screen "fp_motor" 500x500
   on GenerateScreen: "show_tab"(1)
   IOField "I/O field_current" at 172,288 size 68x16; FormatPattern 999.9; Unit  A
      ProcessValue <- ".AO1b"
      Visibility <- ".FP_SHOW.AI1"
   IOField "I/O field_power" at 172,308 size 68x16; FormatPattern 999.9; Unit  kW
      ProcessValue <- ".AO2b"
      Visibility <- ".FP_SHOW.AI2"
   IOField "I/O field_rpm" at 172,328 size 68x16; FormatPattern 9999; Unit  rpm
      ProcessValue <- ".AO3b"
      Visibility <- ".FP_SHOW.AI3"
   IOField "I/O field_set_spd" at 84,356 size 68x16; FormatPattern 999.9; Unit  %
      ProcessValue <- ".SPSET"
      Visibility <- ".FP_SHOW.SP"
   Button "btn_md_auto" at 20,193 size 80x30; TextOff 'Auto'; Authorization "Operate"
      ObjectEnable <- ".FP_DIM.Auto"
      Visibility <- ".FP_SHOW.PB_Auto"
      Appearance <- ".ModePointer"
      on Click: SetBit(".FP_CMD.Auto")
   TextField "cntrl_box_cntrl_head" at 12,68 size 86x22; Text 'Start/Stop'
   Button "btn_md_loc" at 107,193 size 80x30; TextOff 'Local'; Authorization "Operate"
      ObjectEnable <- ".FP_DIM.Local"
      Visibility <- ".FP_SHOW.PB_Local"
      Appearance <- ".ModePointer"
      on Click: SetBit(".FP_CMD.Local")
   TextField "cntrl_box_model_head" at 12,164 size 49x22; Text 'Mode'
   Button "btn_md_man" at 195,193 size 80x30; TextOff 'Man'; Authorization "Operate"
      ObjectEnable <- ".FP_DIM.Manual"
      Visibility <- ".FP_SHOW.PB_Manual"
      Appearance <- ".ModePointer"
      on Click: SetBit(".FP_CMD.Manual")
   TextField "cntrl_box_am_text" at 20,288 size 47x17; Text 'Current'
      Visibility <- ".FP_SHOW.AI1"
   TextField "cntrl_box_am_text_1" at 20,308 size 38x17; Text 'Power'
      Visibility <- ".FP_SHOW.AI2"
   TextField "cntrl_box_model_head_1" at 12,260 size 162x22; Text 'Analog Measurment'
   TextField "cntrl_box_am_text_2" at 20,328 size 27x17; Text 'RPM'
      Visibility <- ".FP_SHOW.AI3"
   TextField "cntrl_box_am_text_3" at 20,355 size 16x17; Text 'SP'
      Visibility <- ".FP_SHOW.SP"
   IOField "I/O field_current_1" at 84,288 size 68x16; FormatPattern 999.9; Unit  %
      ProcessValue <- ".AO1a"
      Visibility <- ".FP_SHOW.AI1"
   IOField "I/O field_power_1" at 84,308 size 68x16; FormatPattern 999.9; Unit  %
      ProcessValue <- ".AO2a"
      Visibility <- ".FP_SHOW.AI2"
   IOField "I/O field_rpm_1" at 84,328 size 68x16; FormatPattern 999.9; Unit  %
      ProcessValue <- ".AO3a"
      Visibility <- ".FP_SHOW.AI3"
   Button "btn_satrt" at 20,100 size 80x30; TextOff 'Start'; Authorization "Operate"
      Visibility <- ".FP_SHOW.PB_Start1"
      ObjectEnable <- ".FP_DIM.Start1"
      on Click: SetBit(".FP_CMD.Start1")
   Button "btn_stop" at 300,100 size 80x30; TextOff 'Stop'; Authorization "Operate"
      Visibility <- ".FP_SHOW.PB_Stop"
      ObjectEnable <- ".FP_DIM.Stop"
      on Click: SetBit(".FP_CMD.Stop")
   TextField "header_txt" at 8,8 size 396x21; Text 'HEADER'
      Text <- ".DefaultText"
   SymbolicIOField "status I/O field_1" at 8,32 size 396x32; TextOn '1'; TextOff '0'; TextList "motor_status"
      ProcessValue <- ".StatusWork"
      Appearance <- ".StatusWork"
   SymbolicIOField "status I/O field_2" at 468,4 size 24x24; TextOn '1'; TextOff '0'; TextList "mode_l"
      ProcessValue <- ".ModePointer"
      Appearance <- ".ModePointer"
   Button "bt_tab_1" at 412,76 size 80x28; TextOff 'Control'
      on Click: "show_tab"(1)
   Button "bt_tab_3" at 412,139 size 80x28; TextOff 'Input'
      on Click: "show_tab"(3)
   Button "bt_tab_4" at 412,171 size 80x28; TextOff 'Output'
      on Click: "show_tab"(4)
   Button "bt_tab_5" at 412,203 size 80x28; TextOff 'Timers'
      on Click: "show_tab"(5)
   Button "bt_tab_6" at 412,235 size 80x28; TextOff 'Analog'
      on Click: "show_tab"(6)
   Button "bt_tab_7" at 412,267 size 80x28; TextOff 'Point para'
      on Click: "show_tab"(7)
   Button "bt_tab_8" at 412,299 size 80x28; TextOff 'Config'
      on Click: "show_tab"(8)
   Button "bt_tab_11" at 412,396 size 80x28; TextOff 'Info'
      on Click: "show_tab"(11)
   Button "bt_tab_12" at 412,428 size 80x28; TextOff 'Motion'
      on Click: "show_tab"(12)
      Visibility <- ".FP_SHOW.MD"
   Button "bt_tab_9" at 412,331 size 80x28; TextOff 'Config2'
      on Click: "show_tab"(9)
   Button "bt_tab_10" at 412,364 size 80x28; TextOff 'Diag'
      on Click: "show_tab"(10)
   Button "bt_tab_2" at 412,108 size 80x28; TextOff 'Interlock'
      on Click: "show_tab"(2)
   TextField "input_head" at 15,68 size 38x19; Text 'Input'
   TextField "input_rdy" at 24,96 size 200x20; Text 'RDY Ready'
   TextField "input_mcc" at 24,120 size 200x20; Text 'MCC MCC Ready'
   TextField "input_ovl" at 24,144 size 200x20; Text 'OVL Overload'
   TextField "input_ret1" at 24,168 size 200x20; Text 'RET1 Return'
   TextField "input_lstr1" at 24,192 size 200x20; Text 'LSTR1 Local Start'
   TextField "input_lstp" at 24,216 size 200x20; Text 'LSTP Local Stop'
   TextField "input_rem" at 24,240 size 200x20; Text 'REM Remote'
   TextField "input_ssw" at 24,264 size 200x20; Text 'SSW Safety Switch'
   TextField "input_es" at 24,288 size 200x20; Text 'ES Excessive Strt'
   TextField "input_tfaa" at 224,96 size 180x20; Text 'TFA Thermistor'
   TextField "input_drdy" at 225,120 size 180x20; Text 'DRDY Drv/MCC Rdy'
   TextField "input_stall" at 225,144 size 180x20; Text 'STALL Mtr Stalled'
   TextField "input_earth" at 225,168 size 180x20; Text 'EARTH Earth Fault'
   TextField "input_ubal" at 225,192 size 180x20; Text 'UBAL Crnt Unbal'
   TextField "input_gfa" at 224,216 size 180x20; Text 'GFA Gen Fault'
   TextField "input_gwa" at 224,240 size 180x20; Text 'GWA Gen Warn'
   TextField "input_busf" at 224,264 size 180x20; Text 'BUSF Bus Fault'
   TextField "input_dopr" at 224,288 size 180x20; Text 'DOPR Oper Posit'
   TextField "input_dtst" at 224,312 size 180x20; Text 'DTEST Test Pos'
   TextField "input_ack" at 224,336 size 180x20; Text 'ACK Reset Ack'
   TextField "input_head_1" at 202,68 size 106x19; Text 'Extend Input'
   TextField "input_head_2" at 13,352 size 96x19; Text 'Miscellaneous'
   TextField "input_sel" at 24,373 size 180x20; Text 'SEL Select'
   TextField "input_astr" at 24,396 size 200x20; Text 'ASTR Auto Start Req'
   IOField "status_bit_1g_0r_3" at 72,96 size 20x20; FormatPattern 1; Unit  
      ProcessValue <- ".DI.RDY"
      Appearance <- ".DI.RDY"
   IOField "status_bit_1g_0r_2" at 72,120 size 20x20; FormatPattern 1; Unit  
      ProcessValue <- ".DI.MCC"
      Appearance <- ".DI.MCC"
   IOField "status_bit_1g_0r_4" at 72,144 size 20x20; FormatPattern 1; Unit  
      ProcessValue <- ".DI.OVL"
      Appearance <- ".DI.OVL"
   IOField "status_bit_1grn_0gry_5" at 72,168 size 20x20; FormatPattern 1; Unit  
      ProcessValue <- ".DI.RET1"
      Appearance <- ".DI.RET1"
   IOField "status_bit_1grn_0gry_1" at 72,192 size 20x20; FormatPattern 1; Unit  
      ProcessValue <- ".DI.LSTR1"
      Appearance <- ".DI.LSTR1"
   IOField "status_bit_1g_0r_5" at 72,216 size 20x20; FormatPattern 1; Unit  
      ProcessValue <- ".DI.LSTP"
      Appearance <- ".DI.LSTP"
   IOField "status_bit_1g_0r_6" at 72,240 size 20x20; FormatPattern 1; Unit  
      ProcessValue <- ".DI.REM"
      Appearance <- ".DI.REM"
   IOField "status_bit_1g_0r_7" at 72,264 size 20x20; FormatPattern 1; Unit  
      Appearance <- ".DI.SSW"
      ProcessValue <- ".DI.SSW"
   IOField "status_bit_1g_0g_8" at 72,288 size 20x20; FormatPattern 1; Unit  
      ProcessValue <- ".DI.ES"
   IOField "status_bit_1g_0r_1" at 276,92 size 20x20; FormatPattern 1; Unit  
      ProcessValue <- ".DI.TFA"
      Appearance <- ".DI.TFA"
   IOField "status_bit_1g_0r_8" at 276,120 size 20x20; FormatPattern 1; Unit  
      ProcessValue <- ".DI.DRDY"
      Appearance <- ".DI.DRDY"
   IOField "status_bit_1g_0r_9" at 276,144 size 20x20; FormatPattern 1; Unit  
      ProcessValue <- ".DI.STALL"
      Appearance <- ".DI.STALL"
   IOField "status_bit_1g_0r_10" at 276,168 size 20x20; FormatPattern 1; Unit  
      ProcessValue <- ".DI.EARTH"
      Appearance <- ".DI.EARTH"
   IOField "status_bit_1g_0r_11" at 276,192 size 20x20; FormatPattern 1; Unit  
      ProcessValue <- ".DI.UBAL"
      Appearance <- ".DI.UBAL"
   IOField "status_bit_1g_0r_12" at 276,216 size 20x20; FormatPattern 1; Unit  
      ProcessValue <- ".DI.GFA"
      Appearance <- ".DI.GFA"
   IOField "status_bit_1g_0r_13" at 276,240 size 20x20; FormatPattern 1; Unit  
      ProcessValue <- ".DI.GWA"
      Appearance <- ".DI.GWA"
   IOField "status_bit_1g_0r_14" at 276,264 size 20x20; FormatPattern 1; Unit  
      ProcessValue <- ".DI.BUSF"
      Appearance <- ".DI.BUSF"
   IOField "status_bit_1g_0r_15" at 276,288 size 20x20; FormatPattern 1; Unit  
      ProcessValue <- ".DI.DOPR"
      Appearance <- ".DI.DOPR"
   IOField "status_bit_1grn_0gry_2" at 276,336 size 20x20; FormatPattern 1; Unit  
      ProcessValue <- ".DI.ACK"
      Appearance <- ".DI.ACK"
   IOField "status_bit_1red_0gry_3" at 276,312 size 20x20; FormatPattern 1; Unit  
      ProcessValue <- ".DI.DTEST"
      Appearance <- ".DI.DTEST"
   IOField "status_bit_1grn_0gry_3" at 72,373 size 20x20; FormatPattern 1; Unit  
      ProcessValue <- ".DI.SEL"
      Appearance <- ".DI.SEL"
   IOField "status_bit_1grn_0gry_4" at 72,396 size 20x20; FormatPattern 1; Unit  
      ProcessValue <- ".DI.ASTR"
      Appearance <- ".DI.ASTR"
   TextField "output_head_3" at 15,68 size 49x19; Text 'Output'
   TextField "output_ok_1" at 24,96 size 200x20; Text 'OK OK'
   TextField "output_sack_1" at 24,120 size 200x20; Text 'SACK Start Ack'
   TextField "output__rd1_1" at 24,144 size 200x20; Text 'RD1 Run Delay'
   TextField "output_run_1" at 24,168 size 200x20; Text 'RUN Run'
   TextField "output_con1_1" at 24,192 size 200x20; Text 'CON1 Command'
   TextField "input_tfaa_1" at 224,96 size 180x20; Text 'LOC Local'
   TextField "input_drdy_1" at 225,120 size 180x20; Text 'AUT Auto'
   TextField "input_stall_1" at 225,144 size 180x20; Text 'MAN Manual'
   TextField "input_earth_1" at 225,168 size 180x20; Text 'SS Single Strt'
   TextField "input_ubal_1" at 225,192 size 180x20; Text 'TESTP Test Pem'
   TextField "input_gfa_1" at 224,216 size 180x20; Text 'RES Reset'
   TextField "input_gwa_1" at 224,240 size 180x20; Text 'ASTW Start Warn'
   TextField "Output_head_4" at 202,68 size 114x19; Text 'Output Modes'
   TextField "output_head_5" at 13,291 size 38x19; Text 'Reset'
   IOField "status_bit_1g_0r_16" at 72,96 size 20x20; FormatPattern 1; Unit  
      ProcessValue <- ".DQ.OK"
      Appearance <- ".DQ.OK"
   IOField "status_bit_1g_0r_17" at 72,120 size 20x20; FormatPattern 1; Unit  
      ProcessValue <- ".DQ.SACK"
      Appearance <- ".DQ.SACK"
   IOField "status_bit_1g_0r_18" at 72,144 size 20x20; FormatPattern 1; Unit  
      ProcessValue <- ".DQ.RD1"
      Appearance <- ".DQ.RD1"
   IOField "status_bit_1grn_0gry_6" at 72,168 size 20x20; FormatPattern 1; Unit  
      ProcessValue <- ".DQ.RUN1"
      Appearance <- ".DQ.RUN1"
   IOField "status_bit_1grn_0gry_7" at 72,192 size 20x20; FormatPattern 1; Unit  
      ProcessValue <- ".DQ.CON1"
      Appearance <- ".DQ.CON1"
   IOField "status_bit_1g_0r_22" at 276,92 size 20x20; FormatPattern 1; Unit  
      ProcessValue <- ".DQ.LOC"
      Appearance <- ".DQ.LOC"
   IOField "status_bit_1g_0r_23" at 276,120 size 20x20; FormatPattern 1; Unit  
      ProcessValue <- ".DQ.AUT"
      Appearance <- ".DQ.AUT"
   IOField "status_bit_1g_0r_24" at 276,144 size 20x20; FormatPattern 1; Unit  
      ProcessValue <- ".DQ.MAN"
      Appearance <- ".DQ.MAN"
   IOField "status_bit_1g_0r_25" at 276,168 size 20x20; FormatPattern 1; Unit  
      ProcessValue <- ".DQ.SS"
      Appearance <- ".DQ.SS"
   IOField "status_bit_1g_0r_26" at 276,192 size 20x20; FormatPattern 1; Unit  
      ProcessValue <- ".DQ.TESTP"
      Appearance <- ".DQ.TESTP"
   IOField "status_bit_1g_0r_27" at 276,216 size 20x20; FormatPattern 1; Unit  
      ProcessValue <- ".DQ.RES"
      Appearance <- ".DQ.RES"
   IOField "status_bit_1g_0r_28" at 276,240 size 20x20; FormatPattern 1; Unit  
      ProcessValue <- ".DQ.ASTW"
      Appearance <- ".DQ.ASTW"
   Button "btn_reset" at 172,318 size 80x30; TextOff 'Reset'
      on Click: SetBit(".FP_CMD.Reset")
      ObjectEnable <- ".FP_DIM.Reset"
      Visibility <- ".FP_SHOW.PB_Reset"
   TextField "output_head_1" at 16,69 size 49x19; Text 'Timers'
   TextField "timers_text" at 24,96 size 100x20; Text 'Delay Start'
   IOField "delay_start_tm_sp" at 132,96 size 60x20; Authorization "User administration"; FormatPattern 9999; Unit  s
      ProcessValue <- ".FP_PARM.DelayStart_Pre"
   TextField "timers_text_1" at 24,120 size 100x20; Text 'Return M Tm'
   TextField "timers_text_2" at 24,144 size 100x20; Text 'Delayed Run'
   TextField "timers_text_3" at 24,168 size 100x20; Text 'Delayed Stop'
   TextField "timers_text_4" at 24,192 size 100x20; Text 'Start Warning'
   IOField "return_tm_sp" at 132,120 size 60x20; Authorization "User administration"; FormatPattern 9999; Unit  s
      ProcessValue <- ".FP_PARM.ReturnMon_Pre"
   IOField "delayed_run_tm_sp" at 132,144 size 60x20; Authorization "User administration"; FormatPattern 9999; Unit  s
      ProcessValue <- ".FP_PARM.RunDelay1_Pre"
   IOField "delay_stop_tm_sp" at 132,168 size 60x20; Authorization "User administration"; FormatPattern 999; Unit  s
      ProcessValue <- ".FP_PARM.DelayStop_Pre"
   IOField "delay_startsrm_tm_sp" at 132,192 size 60x20; Authorization "User administration"; FormatPattern 999; Unit  s
      ProcessValue <- ".FP_PARM.StartWarn_Pre"
   TextField "output_head_2" at 16,69 size 58x19; Text 'Current'
   TextField "analog_text_1" at 24,115 size 100x20; Text 'Minimum'
   IOField "ai1_min_sp" at 132,115 size 60x20; Authorization "User administration"; FormatPattern 9999.9; Unit  
      ProcessValue <- ".FP_PARM.AI1_Min"
   TextField "analog_text_2" at 147,93 size 33x17; Text 'Input'
   TextField "analog_text_3" at 223,93 size 44x17; Text 'Output'
   TextField "analog_text_4" at 303,93 size 36x17; Text 'Out:A'
   IOField "ao1a_min_sp" at 212,115 size 60x20; Authorization "User administration"; FormatPattern 9999.9; Unit  
      ProcessValue <- ".FP_PARM.AO1a_Min"
   IOField "ao1b_min_sp" at 292,115 size 60x20; Authorization "User administration"; FormatPattern 9999.9; Unit  
      ProcessValue <- ".FP_PARM.AO1b_Min"
   TextField "analog_text_5" at 24,139 size 100x20; Text 'Maximum'
   IOField "ai1_max_sp_1" at 132,139 size 60x20; Authorization "User administration"; FormatPattern 9999.9; Unit  
      ProcessValue <- ".FP_PARM.AI1_Max"
   IOField "ao1a_max_sp_1" at 212,139 size 60x20; Authorization "User administration"; FormatPattern 9999.9; Unit  
      ProcessValue <- ".FP_PARM.AO1a_Max"
   IOField "ao1b_max_sp_1" at 292,139 size 60x20; Authorization "User administration"; FormatPattern 9999.9; Unit  
      ProcessValue <- ".FP_PARM.AO1b_Max"
   IOField "ai1" at 132,167 size 60x20; FormatPattern 9999.9; Unit  
      ProcessValue <- ".AI1"
   IOField "ao1a" at 212,167 size 60x20; FormatPattern 9999.9; Unit  %
      ProcessValue <- ".AO1a"
   IOField "ao1b" at 292,167 size 60x20; FormatPattern 9999.9; Unit  A
      ProcessValue <- ".AO1b"
   TextField "output_head_6" at 15,196 size 49x19; Text 'Power'
   TextField "analog_text_6" at 23,243 size 100x20; Text 'Minimum'
   IOField "ai2_min_sp_1" at 131,243 size 60x20; Authorization "User administration"; FormatPattern 9999.9; Unit  
      ProcessValue <- ".FP_PARM.AI2_Min"
   TextField "analog_text_7" at 146,221 size 33x17; Text 'Input'
   TextField "analog_text_8" at 222,221 size 44x17; Text 'Output'
   TextField "analog_text_9" at 302,221 size 36x17; Text 'Out:A'
   IOField "ao2a_min_sp_1" at 211,243 size 60x20; Authorization "User administration"; FormatPattern 9999.9; Unit  
      ProcessValue <- ".FP_PARM.AO2a_Min"
   IOField "ao2b_min_sp_1" at 291,243 size 60x20; Authorization "User administration"; FormatPattern 9999.9; Unit  
      ProcessValue <- ".FP_PARM.AO2b_Min"
   TextField "analog_text_10" at 23,267 size 100x20; Text 'Maximum'
   IOField "ai2_max_sp_2" at 131,267 size 60x20; Authorization "User administration"; FormatPattern 9999.9; Unit  
      ProcessValue <- ".FP_PARM.AI2_Max"
   IOField "ao2a_max_sp_2" at 211,267 size 60x20; Authorization "User administration"; FormatPattern 9999.9; Unit  
      ProcessValue <- ".FP_PARM.AO2a_Max"
   IOField "ao2b_max_sp_2" at 291,267 size 60x20; Authorization "User administration"; FormatPattern 9999.9; Unit  
      ProcessValue <- ".FP_PARM.AO2b_Max"
   IOField "ai2_1" at 131,295 size 60x20; FormatPattern 9999.9; Unit  
      ProcessValue <- ".AI2"
   IOField "ao2a_1" at 211,295 size 60x20; FormatPattern 9999.9; Unit  %
      ProcessValue <- ".AO2a"
   IOField "ao2b_1" at 291,295 size 60x20; FormatPattern 9999.9; Unit  A
      ProcessValue <- ".AO2b"
   TextField "output_head_7" at 14,324 size 36x19; Text 'RPM'
   TextField "analog_text_11" at 23,372 size 100x20; Text 'Minimum'
   IOField "ai3_min_sp_2" at 131,372 size 60x20; Authorization "User administration"; FormatPattern 9999.9; Unit  
      ProcessValue <- ".FP_PARM.AI3_Min"
   TextField "analog_text_12" at 145,350 size 33x17; Text 'Input'
   TextField "analog_text_13" at 221,350 size 44x17; Text 'Output'
   TextField "analog_text_14" at 301,350 size 36x17; Text 'Out:A'
   IOField "ao3a_min_sp_2" at 211,372 size 60x20; Authorization "User administration"; FormatPattern 9999.9; Unit  
      ProcessValue <- ".FP_PARM.AO3a_Min"
   IOField "ao3b_min_sp_2" at 291,372 size 60x20; Authorization "User administration"; FormatPattern 9999.9; Unit  
      ProcessValue <- ".FP_PARM.AO3b_Min"
   TextField "analog_text_15" at 23,396 size 100x20; Text 'Maximum'
   IOField "ai3_max_sp_3" at 131,396 size 60x20; Authorization "User administration"; FormatPattern 9999.9; Unit  
      ProcessValue <- ".FP_PARM.AI3_Max"
   IOField "ao3a_max_sp_3" at 211,396 size 60x20; Authorization "User administration"; FormatPattern 9999.9; Unit  
      ProcessValue <- ".FP_PARM.AO3a_Max"
   IOField "ao3b_max_sp_3" at 291,396 size 60x20; Authorization "User administration"; FormatPattern 9999.9; Unit  
      ProcessValue <- ".FP_PARM.AO3b_Max"
   IOField "ai3_2" at 131,424 size 60x20; FormatPattern 9999.9; Unit  
      ProcessValue <- ".AI3"
   IOField "ao3a_2" at 211,424 size 60x20; FormatPattern 9999.9; Unit  %
      ProcessValue <- ".AO3a"
   IOField "ao3b_2" at 291,424 size 60x20; FormatPattern 9999.9; Unit  A
      ProcessValue <- ".AO3b"
   TextField "output_head_8" at 20,70 size 58x19; Text 'Current'
   CheckBox "Check box_1" at 28,96 size 180x20; Text0 'Alarm Supression'; Authorization "User administration"
   TextField "output_head_9" at 20,70 size 74x19; Text 'Unit Type'
   CheckBox "cb_Type_Indication" at 12,144 size 180x20; Text0 'Indication'; Authorization "User administration"
      ProcessValue <- ".FP_SEL.Type_Indication"
   OptionGroup "op_Type_Unimotor" at 12,96 size 180x20; Text0 'Uni directional motor'; Authorization "User administration"
      ProcessValue <- ".FP_SEL.Type_Unimotor"
   OptionGroup "op_Type_Bimotor" at 12,120 size 180x20; Text0 'Bi directional motor'; Authorization "User administration"
      ProcessValue <- ".FP_SEL.Type_Bimotor"
   CheckBox "cb_OutOfSevice" at 12,168 size 180x20; Text0 'Out of Sevices'; Authorization "User administration"
      ProcessValue <- ".FP_SEL.OutOfSevice"
   TextField "output_head_10" at 188,70 size 164x19; Text 'Start Warning Enable'
   CheckBox "cb_STW_Single" at 200,96 size 180x20; Text0 'Single Start'; Authorization "User administration"
      ProcessValue <- ".FP_SEL.STW_Single"
   CheckBox "cb_STW_Manual" at 200,120 size 180x20; Text0 'Manual'; Authorization "User administration"
      ProcessValue <- ".FP_SEL.STW_Manual"
   CheckBox "cb_STW_AutoStart" at 200,144 size 188x20; Text0 'Intrval Str (Auto Start)'; Authorization "User administration"
      ProcessValue <- ".FP_SEL.STW_AutoStart"
   CheckBox "cb_STW_Loca" at 200,168 size 188x20; Text0 'Local'; Authorization "User administration"
      ProcessValue <- ".FP_SEL.STW_Local"
   TextField "output_head_11" at 20,198 size 107x19; Text 'Alarm Handing'
   TextField "output_head_12" at 188,198 size 112x19; Text 'Enable Modes'
   CheckBox "Check box_8" at 12,224 size 180x20; Text0 'Warning Drive'; Authorization "User administration"
      ProcessValue <- ".FP_SEL.WarningDrive"
   CheckBox "Check box_9" at 12,248 size 180x20; Text0 'Sup by Parent Grp'; Authorization "User administration"
      ProcessValue <- ".FP_SEL.ParentSupress"
   CheckBox "Check box_10" at 12,272 size 188x20; Text0 'Pass Status to Par Grp'; Authorization "User administration"
      ProcessValue <- ".FP_SEL.ParentCollection"
   CheckBox "Check box_11" at 200,224 size 180x20; Text0 'Automatic'; Authorization "User administration"
      ProcessValue <- ".FP_EN.Mode_Auto"
   CheckBox "Check box_12" at 200,248 size 180x20; Text0 'Manual'; Authorization "User administration"
      ProcessValue <- ".FP_EN.Mode_Man"
   CheckBox "Check box_13" at 200,272 size 188x20; Text0 'Local'; Authorization "User administration"
      ProcessValue <- ".FP_EN.Mode_Loc"
   CheckBox "Check box_14" at 200,296 size 188x20; Text0 'Single Start FP'; Authorization "User administration"
      ProcessValue <- ".FP_EN.Mode_SS_FP"
   CheckBox "Check box_15" at 200,320 size 188x20; Text0 'Single Start Filed'; Authorization "User administration"
      ProcessValue <- ".FP_EN.Mode_SS_Field"
   CheckBox "Check box_16" at 200,344 size 188x20; Text0 'Test mode'; Authorization "User administration"
      ProcessValue <- ".FP_EN.Mode_Test"
   TextField "output_head_13" at 20,296 size 111x19; Text 'Enable Features'
   CheckBox "Check box_17" at 12,320 size 180x20; Text0 'Motion'; Authorization "User administration"
      ProcessValue <- ".FP_SEL.MD"
   CheckBox "Check box_18" at 12,344 size 180x20; Text0 'Motor Starter'; Authorization "User administration"
      ProcessValue <- ".FP_SEL.MotorStarter"
   CheckBox "Check box_19" at 12,368 size 188x20; Text0 'Quick Stop frm Unit'; Authorization "User administration"
      ProcessValue <- ".FP_EN.PB_QStop"
   CheckBox "Check box_20" at 12,392 size 188x20; Text0 'Reset Btn on Faceplate'; Authorization "User administration"
      ProcessValue <- ".FP_SHOW.PB_Reset"
   CheckBox "Check box_21" at 12,440 size 180x20; Text0 'Inch in Man Mode'; Authorization "User administration"
      ProcessValue <- ".FP_SEL.INCH_Man"
   CheckBox "Check box_22" at 12,464 size 180x20; Text0 'Inch in Loc Mode'; Authorization "User administration"
      ProcessValue <- ".FP_SEL.INCH_Loc"
   CheckBox "Check box_23" at 200,392 size 180x20; Text0 'Current'; Authorization "User administration"
      ProcessValue <- ".FP_SHOW.AI1"
   CheckBox "Check box_24" at 200,416 size 180x20; Text0 'Power'; Authorization "User administration"
      ProcessValue <- ".FP_SHOW.AI2"
   CheckBox "Check box_25" at 200,440 size 188x20; Text0 'RPM'; Authorization "User administration"
      ProcessValue <- ".FP_SHOW.AI3"
   CheckBox "Check box_26" at 200,464 size 188x20; Text0 'SP'; Authorization "User administration"
      ProcessValue <- ".FP_SHOW.SP"
   TextField "output_head_16" at 206,367 size 157x19; Text 'Display Analog Values'
   TextField "output_head_17" at 20,416 size 105x19; Text 'Inching Enable'
   TextField "output_head_14" at 20,70 size 98x19; Text 'Displat Inputs'
   CheckBox "cb_Type_Indication_1" at 204,300 size 100x20; Text0 'ASTRT'; Authorization "User administration"
      ProcessValue <- ".FP_SHOW.ASTR"
   CheckBox "cb_Type_Indication_2" at 16,100 size 100x192; Text0 'AI1'; Text1 'AI2'; Text2 'AI3'; Text3 'SP'; Text4 'MCC'; Text5 'RDY'; Text6 'OVL'; Text7 'LSTP'; Authorization "User administration"
      ProcessValue <- ".FP_SHOW.B1"
   CheckBox "cb_Type_Indication_3" at 108,100 size 100x192; Text6 'EARTH'; Text7 'UBAL'; Text4 'DRDY'; Text5 'STALL'; Text2 'ES'; Text3 'TFA'; Text0 'REM'; Text1 'SSW'; Authorization "User administration"
      ProcessValue <- ".FP_SHOW.B2"
   CheckBox "cb_Type_Indication_4" at 204,100 size 100x192; Text6 'LSTR1'; Text4 'DTEST'; Text5 'ACK'; Text2 'BUSF'; Text3 'DOPR'; Text0 'GFA'; Text1 'GWA'; Text7 'LSTR2'; Authorization "User administration"
      ProcessValue <- ".FP_SHOW.B3"
   TextField "output_head_15" at 15,68 size 114x19; Text 'PLC Subroutine'
   TextField "text_16" at 24,92 size 100x20; Text 'SubRoutine'
   TextField "text_1" at 24,120 size 100x20; Text 'Version'
   IOField "iof_vers" at 136,120 size 60x20; FormatPattern 9999; Unit  
      ProcessValue <- "[0]"
   TextField "text_2" at 24,148 size 100x20; Text 'Build'
   IOField "iof_build" at 136,148 size 60x20; FormatPattern 9999; Unit  
      ProcessValue <- "[1]"
   TextField "text_3" at 24,176 size 100x20; Text 'IOSys'
   TextField "output_head_18" at 212,68 size 129x19; Text 'Program Status'
   TextField "text_4" at 226,92 size 100x20; Text 'State Pointer'
   IOField "iof_state_pointer" at 338,92 size 60x20; FormatPattern 9999; Unit  
      ProcessValue <- ".BlockInfo[2]"
   TextField "text_5" at 227,120 size 100x20; Text 'State Pointer_Prev'
   IOField "iof_state_pointer_prev" at 339,120 size 60x20; FormatPattern 9999; Unit  
      ProcessValue <- ".BlockInfo[3]"
   TextField "output_head_19" at 16,228 size 106x19; Text 'PLC Reference'
   TextField "text_6" at 24,256 size 100x20; Text 'DB'
   IOField "iof_db" at 136,256 size 60x20; FormatPattern 9999; Unit  
      ProcessValue <- ".BlockInfo[4]"
   TextField "output_head_20" at 16,292 size 51x19; Text 'EcsRef'
   TextField "output_head_21" at 16,412 size 79x19; Text 'ParentInfo'
   TextField "text_7" at 24,320 size 100x20; Text 'FP Name'
   TextField "text_8" at 24,348 size 100x20; Text 'Blk Alg Ver'
   TextField "text_9" at 24,376 size 100x20; Text 'Status Alg Ver'
   IOField "parent_info" at 24,440 size 380x20; FormatPattern *; Unit  
      ProcessValue <- ".ParentInfo"
   TextField "interlockl_head_1" at 16,68 size 93x22; Text 'Interlocking'
   TextField "interlockl_head_2" at 12,225 size 174x22; Text 'Sequence Interlocking'
   TextField "interlockl_head_3" at 12,383 size 175x22; Text 'Sequence Stop Enable'
   TextField "interlock_1" at 28,100 size 140x20; Text 'Interlock 1'
      Text <- ".INTL01.DefaultText"
      Visibility <- ".INTL01"
   TextField "interlock_2" at 28,128 size 140x20; Text 'Interlock 2'
      Text <- ".INTL02.DefaultText"
      Visibility <- ".INTL04"
   TextField "interlock_3" at 28,156 size 140x20; Text 'Interlock 3'
      Text <- ".INTL03.DefaultText"
      Visibility <- ".INTL04"
   TextField "interlock_4" at 28,184 size 140x20; Text 'Interlock 4'
      Text <- ".INTL04.DefaultText"
      Visibility <- ".INTL04"
   TextField "STRT_1" at 28,256 size 140x20; Text 'Interlock 1'
      Visibility <- ".STR01"
      Text <- ".STR01.DefaultText"
   TextField "STRT_2" at 28,284 size 140x20; Text 'Interlock 2'
      Visibility <- ".STR02"
      Text <- ".STR02.DefaultText"
   TextField "STRT_3" at 28,312 size 140x20; Text 'Interlock 3'
      Visibility <- ".STR03"
      Text <- ".STR03.DefaultText"
   TextField "STRT_4" at 28,340 size 140x20; Text 'Interlock 4'
      Visibility <- ".STR04"
      Text <- ".STR04.DefaultText"
   SymbolicIOField "int_01" at 164,100 size 45x20; TextOn '1'; TextOff '0'; TextList "interlock_status_byte"
      ProcessValue <- ".INTL01"
      Appearance <- ".INTL01"
      Visibility <- ".INTL01"
   SymbolicIOField "int_2" at 164,128 size 45x20; TextOn '1'; TextOff '0'; TextList "interlock_status_byte"
      Visibility <- ".INTL02"
      ProcessValue <- ".INTL02"
      Appearance <- ".INTL02"
   SymbolicIOField "int_1" at 163,156 size 45x20; TextOn '1'; TextOff '0'; TextList "interlock_status_byte"
      ProcessValue <- ".INTL03"
      Visibility <- ".INTL03"
      Appearance <- ".INTL03"
   SymbolicIOField "int_3" at 164,184 size 45x20; TextOn '1'; TextOff '0'; TextList "interlock_status_byte"
      ProcessValue <- ".INTL04"
      Visibility <- ".INTL04"
      Appearance <- ".INTL04"
   TextField "interlock_5" at 221,100 size 140x20; Text 'Interlock 5'
      Text <- ".INTL05.DefaultText"
      Visibility <- ".INTL05"
   TextField "interlock_6" at 221,128 size 140x20; Text 'Interlock 6'
      Text <- ".INTL06.DefaultText"
      Visibility <- ".INTL06"
   TextField "interlock_7" at 221,156 size 140x20; Text 'Interlock 7'
      Text <- ".INTL07.DefaultText"
      Visibility <- ".INTL07"
   TextField "interlock_8" at 221,184 size 140x20; Text 'Interlock 8'
      Text <- ".INTL08.DefaultText"
      Visibility <- ".INTL08"
   SymbolicIOField "int_4" at 357,100 size 45x20; TextOn '1'; TextOff '0'; TextList "interlock_status_byte"
      Visibility <- ".INTL05"
      Appearance <- ".INTL05"
      ProcessValue <- ".INTL05"
   SymbolicIOField "int_5" at 357,128 size 45x20; TextOn '1'; TextOff '0'; TextList "interlock_status_byte"
      Visibility <- ".INTL06"
      Appearance <- ".INTL06"
      ProcessValue <- ".INTL06"
   SymbolicIOField "int_6" at 356,156 size 45x20; TextOn '1'; TextOff '0'; TextList "interlock_status_byte"
      Visibility <- ".INTL07"
      Appearance <- ".INTL07"
      ProcessValue <- ".INTL07"
   SymbolicIOField "int_7" at 357,184 size 45x20; TextOn '1'; TextOff '0'; TextList "interlock_status_byte"
      Visibility <- ".INTL08"
      Appearance <- ".INTL08"
      ProcessValue <- ".INTL08"
   SymbolicIOField "int_8" at 164,256 size 45x20; TextOn '1'; TextOff '0'; TextList "interlock_status_byte"
      Visibility <- ".STR01"
      Appearance <- ".STR01"
      ProcessValue <- ".STR01"
   SymbolicIOField "int_9" at 164,284 size 45x20; TextOn '1'; TextOff '0'; TextList "interlock_status_byte"
      Visibility <- ".STR02"
      Appearance <- ".STR02"
      ProcessValue <- ".STR02"
   SymbolicIOField "int_10" at 164,312 size 45x20; TextOn '1'; TextOff '0'; TextList "interlock_status_byte"
      Visibility <- ".STR03"
      Appearance <- ".STR03"
      ProcessValue <- ".STR03"
   SymbolicIOField "int_11" at 164,340 size 45x20; TextOn '1'; TextOff '0'; TextList "interlock_status_byte"
      Visibility <- ".STR04"
      Appearance <- ".STR04"
      ProcessValue <- ".STR04"
   TextField "STRT_5" at 221,256 size 140x20; Text 'Interlock 5'
      Visibility <- ".STR05"
      Text <- ".STR05.DefaultText"
   TextField "STRT_6" at 221,284 size 140x20; Text 'Interlock 6'
      Visibility <- ".STR06"
      Text <- ".STR05.DefaultText"
   TextField "STRT_7" at 221,312 size 140x20; Text 'Interlock 7'
      Visibility <- ".STR07"
      Text <- ".STR06.DefaultText"
   TextField "STRT_8" at 221,340 size 140x20; Text 'Interlock 8'
      Visibility <- ".STR08"
      Text <- ".STR08.DefaultText"
   SymbolicIOField "int_12" at 357,256 size 45x20; TextOn '1'; TextOff '0'; TextList "interlock_status_byte"
      Visibility <- ".STR05"
      Appearance <- ".STR05"
      ProcessValue <- ".STR05"
   SymbolicIOField "int_13" at 357,284 size 45x20; TextOn '1'; TextOff '0'; TextList "interlock_status_byte"
      Visibility <- ".STR06"
      Appearance <- ".STR06"
      ProcessValue <- ".STR06"
   SymbolicIOField "int_14" at 357,312 size 45x20; TextOn '1'; TextOff '0'; TextList "interlock_status_byte"
      Visibility <- ".STR07"
      Appearance <- ".STR07"
      ProcessValue <- ".STR07"
   SymbolicIOField "int_15" at 357,340 size 45x20; TextOn '1'; TextOff '0'; TextList "interlock_status_byte"
      Visibility <- ".STR08"
      Appearance <- ".STR08"
      ProcessValue <- ".STR08"
   TextField "STP_1" at 24,412 size 140x20; Text 'Interlock 1'
      Text <- ".STP01.DefaultText"
      Visibility <- ".STP01"
   TextField "STP_2" at 24,440 size 140x20; Text 'Interlock 2'
      Text <- ".STP02.DefaultText"
      Visibility <- ".STP02"
   TextField "STP_3" at 24,468 size 140x20; Text 'Interlock 3'
      Text <- ".STP03.DefaultText"
      Visibility <- ".STP03"
   SymbolicIOField "stp_int_1" at 160,412 size 45x20; TextOn '1'; TextOff '0'; TextList "interlock_status_byte"
      Visibility <- ".STP01"
      ProcessValue <- ".STP01"
      Appearance <- ".STP01"
   SymbolicIOField "stp_int_2" at 160,440 size 45x20; TextOn '1'; TextOff '0'; TextList "interlock_status_byte"
      Visibility <- ".STP02"
      ProcessValue <- ".STP01"
      Appearance <- ".STP02"
   SymbolicIOField "stp_int_3" at 160,468 size 45x20; TextOn '1'; TextOff '0'; TextList "interlock_status_byte"
      Visibility <- ".STP03"
      ProcessValue <- ".STP03"
      Appearance <- ".STP03"
   TextField "STP_4" at 220,412 size 140x20; Text 'Interlock 4'
      Visibility <- ".STP04"
      Text <- ".STP04.DefaultText"
   TextField "STP_5" at 220,440 size 140x20; Text 'Interlock 5'
      Visibility <- ".STP05"
      Text <- ".STP05.DefaultText"
   TextField "STP_6" at 220,468 size 140x20; Text 'Interlock 6'
      Visibility <- ".STP06"
      Text <- ".STP06.DefaultText"
   SymbolicIOField "stp_int_4" at 356,412 size 45x20; TextOn '1'; TextOff '0'; TextList "interlock_status_byte"
      Visibility <- ".STP04"
      Appearance <- ".STP04"
      ProcessValue <- ".STP04"
   SymbolicIOField "stp_int_5" at 356,440 size 45x20; TextOn '1'; TextOff '0'; TextList "interlock_status_byte"
      Visibility <- ".STP05"
      Appearance <- ".STP05"
      ProcessValue <- ".STP05"
   SymbolicIOField "stp_int_6" at 356,468 size 45x20; TextOn '1'; TextOff '0'; TextList "interlock_status_byte"
      Visibility <- ".STP06"
      Appearance <- ".STP06"
      ProcessValue <- ".STP06"

screen "Main.screen_window1" 0x0
   Siemens.Simatic.Hmi.Utah.GraphX.HmiScreenItem "Rectangle" at 0,0 size 0x0
   Siemens.Simatic.Hmi.Utah.GraphX.HmiScreenItem "header_txt" at 0,0 size 0x0

screen "fp_valve" 500x500
   on GenerateScreen: "show_tab"(1)
   Button "btn_md_auto" at 20,193 size 80x30; TextOff 'Auto'; Authorization "Operate"
      on Click: SetBit(".FP_CMD.Auto")
      Visibility <- ".FP_SHOW.PB_Auto"
      ObjectEnable <- ".FP_DIM.Auto"
      Appearance <- ".ModePointer"
   TextField "cntrl_box_cntrl_head" at 12,68 size 86x22; Text 'Start/Stop'
   Button "btn_md_loc" at 107,193 size 80x30; TextOff 'Local'; Authorization "Operate"
      on Click: SetBit(".FP_CMD.Local")
      Visibility <- ".FP_SHOW.PB_Local"
      ObjectEnable <- ".FP_DIM.Local"
      Appearance <- ".ModePointer"
   TextField "cntrl_box_model_head" at 12,164 size 49x22; Text 'Mode'
   Button "btn_md_man" at 195,193 size 80x30; TextOff 'Man'; Authorization "Operate"
      on Click: SetBit(".FP_CMD.Manual")
      Visibility <- ".FP_SHOW.PB_Manual"
      ObjectEnable <- ".FP_DIM.Manual"
      Appearance <- ".ModePointer"
   Button "btn_open" at 20,100 size 80x30; TextOff 'Open'; Authorization "Operate"
      on Click: SetBit(".FP_CMD.Start1")
      Visibility <- ".FP_SHOW.PB_Start1"
      ObjectEnable <- ".FP_DIM.Start1"
   Button "btn_close" at 300,100 size 80x30; TextOff 'Close'; Authorization "Operate"
      on Click: SetBit(".FP_CMD.Start2")
      ObjectEnable <- ".FP_DIM.Start2"
      Visibility <- ".FP_SHOW.PB_Start2"
   Button "btn_stop" at 156,128 size 80x30; TextOff 'Stop'; Authorization "Operate"
      on Click: SetBit(".FP_CMD.Stop")
      Visibility <- ".FP_SHOW.PB_Stop"
      ObjectEnable <- ".FP_DIM.Stop"
   TextField "header_txt" at 8,8 size 396x21; Text 'HEADER'
      Text <- ".DefaultText"
   SymbolicIOField "status I/O field_2" at 468,4 size 24x24; TextOn '1'; TextOff '0'; TextList "mode_l"
      ProcessValue <- ".ModePointer"
      Appearance <- ".ModePointer"
   Button "bt_tab_1" at 412,76 size 80x28; TextOff 'Control'
      on Click: "show_tab"(1)
   Button "bt_tab_3" at 412,139 size 80x28; TextOff 'Input'
      on Click: "show_tab"(3)
   Button "bt_tab_4" at 412,171 size 80x28; TextOff 'Output'
      on Click: "show_tab"(4)
   Button "bt_tab_5" at 412,203 size 80x28; TextOff 'Timers'
      on Click: "show_tab"(5)
   Button "bt_tab_7" at 412,234 size 80x28; TextOff 'Point para'
      on Click: "show_tab"(7)
   Button "bt_tab_8" at 412,266 size 80x28; TextOff 'Config'
      on Click: "show_tab"(8)
   Button "bt_tab_11" at 412,330 size 80x28; TextOff 'Info'
      on Click: "show_tab"(11)
   Button "bt_tab_9" at 412,298 size 80x28; TextOff 'Config2'
      on Click: "show_tab"(9)
   Button "bt_tab_2" at 412,108 size 80x28; TextOff 'Interlock'
      on Click: "show_tab"(2)
   SymbolicIOField "status I/O field_1" at 124,32 size 165x29; TextOn '1'; TextOff '0'; TextList "valve_status"
      ProcessValue <- ".StatusWork"
      Appearance <- ".StatusWork"
   TextField "input_head" at 15,68 size 38x19; Text 'Input'
   TextField "input_rdy" at 24,96 size 200x20; Text 'RDY Ready'
   TextField "input_ovl" at 24,120 size 200x20; Text 'OVL Overload'
   TextField "input_lstr1" at 24,144 size 200x20; Text 'LSP1 Lim Pos Open'
   TextField "input_lstp" at 24,168 size 200x20; Text 'LSP2 Lim Pos Close'
   TextField "input_rem" at 24,240 size 200x20; Text 'REM Remote'
   TextField "input_ssw" at 24,264 size 200x20; Text 'SSW Safety Switch'
   TextField "input_drdy" at 225,97 size 180x20; Text 'DRDY Drv/MCC Rdy'
   TextField "input_gfa" at 224,121 size 180x20; Text 'GFA Gen Fault'
   TextField "input_gwa" at 224,145 size 180x20; Text 'GWA Gen Warn'
   TextField "input_busf" at 224,169 size 180x20; Text 'BUSF Bus Fault'
   TextField "input_dtst" at 224,193 size 180x20; Text 'UTEST Test Pos'
   TextField "input_head_1" at 202,68 size 106x19; Text 'Extend Input'
   TextField "input_head_2" at 13,352 size 96x19; Text 'Miscellaneous'
   TextField "input_sel" at 24,376 size 180x20; Text 'SEL Select'
   IOField "status_bit_1g_0r_3" at 72,96 size 20x20; FormatPattern 1; Unit  
      ProcessValue <- ".DI.RDY"
      Appearance <- ".DI.RDY"
   IOField "status_bit_1g_0r_4" at 72,120 size 20x20; FormatPattern 1; Unit  
      ProcessValue <- ".DI.OVL"
      Appearance <- ".DI.OVL"
   IOField "status_bit_1grn_0gry_1" at 72,144 size 20x20; FormatPattern 1; Unit  
      Appearance <- ".DI.LSP1"
      ProcessValue <- ".DI.LSP1"
   IOField "status_bit_1g_0r_5" at 72,168 size 20x20; FormatPattern 1; Unit  
      Appearance <- ".DI.LSP2"
      ProcessValue <- ".DI.LSP2"
   IOField "status_bit_1g_0r_6" at 72,240 size 20x20; FormatPattern 1; Unit  
      ProcessValue <- ".DI.REM"
      Appearance <- ".DI.REM"
   IOField "status_bit_1g_0r_7" at 72,264 size 20x20; FormatPattern 1; Unit  
      ProcessValue <- ".DI.SSW"
      Appearance <- ".DI.SSW"
   IOField "status_bit_1g_0r_8" at 276,97 size 20x20; FormatPattern 1; Unit  
      ProcessValue <- ".DI.DRDY"
      Appearance <- ".DI.DRDY"
   IOField "status_bit_1g_0r_12" at 276,121 size 20x20; FormatPattern 1; Unit  
      ProcessValue <- ".DI.GFA"
      Appearance <- ".DI.GFA"
   IOField "status_bit_1g_0r_13" at 276,145 size 20x20; FormatPattern 1; Unit  
      ProcessValue <- ".DI.GWA"
      Appearance <- ".DI.GWA"
   IOField "status_bit_1g_0r_14" at 276,169 size 20x20; FormatPattern 1; Unit  
      ProcessValue <- ".DI.BUSF"
      Appearance <- ".DI.BUSF"
   IOField "status_bit_1red_0gry_3" at 276,193 size 20x20; FormatPattern 1; Unit  
      ProcessValue <- ".DI.UTEST"
      Appearance <- ".DI.UTEST"
   IOField "status_bit_1grn_0gry_3" at 72,376 size 20x20; FormatPattern 1; Unit  
      ProcessValue <- ".DI.SEL"
      Appearance <- ".DI.SEL"
   TextField "input_head_3" at 202,352 size 92x19; Text 'Indications'
   TextField "input_gfa_2" at 222,375 size 180x20; Text 'PREQ1 Req Open'
   TextField "input_gwa_2" at 222,399 size 180x20; Text 'PREQ2 Req Close'
   IOField "status_bit_1g_0r_1" at 274,375 size 20x20; FormatPattern 1; Unit  
      ProcessValue <- ".DI.PREQ1"
      Appearance <- ".DI.PREQ1"
   IOField "status_bit_1g_0r_2" at 274,399 size 20x20; FormatPattern 1; Unit  
      ProcessValue <- ".DI.PREQ2"
      Appearance <- ".DI.PREQ2"
   TextField "input_dtst_1" at 224,217 size 180x20; Text 'ASK Test Pos'
   IOField "status_bit_1red_0gry_1" at 276,217 size 20x20; FormatPattern 1; Unit  
      ProcessValue <- ".DI.ACK"
      Appearance <- ".DI.ACK"
   TextField "input_lstr1_1" at 24,192 size 200x20; Text 'LSTR1 Loc Str Open'
   TextField "input_lstp_1" at 24,215 size 200x20; Text 'LSTR2 Loc Str Close'
   IOField "status_bit_1grn_0gry_2" at 72,192 size 20x20; FormatPattern 1; Unit  
      Appearance <- ".DI.LSTR1"
      ProcessValue <- ".DI.LSTR1"
   IOField "status_bit_1g_0r_9" at 72,215 size 20x20; FormatPattern 1; Unit  
      ProcessValue <- ".DI.LSTR2"
      Appearance <- ".DI.LSTR2"
   TextField "output_head_3" at 15,68 size 54x19; Text 'Output'
   TextField "output_ok_1" at 24,96 size 200x20; Text 'OK OK'
   TextField "output_sack_1" at 24,120 size 200x20; Text 'SACK Start Ack'
   TextField "output__rd1_1" at 24,144 size 200x20; Text 'POS1 Pos Open'
   TextField "output_run_1" at 24,168 size 200x20; Text 'POS2 Pos Close'
   TextField "output_con1_1" at 24,192 size 200x20; Text 'CON1 Cmd Open'
   TextField "input_tfaa_1" at 224,96 size 180x20; Text 'LOC Local'
   TextField "input_drdy_1" at 225,120 size 180x20; Text 'AUT Auto'
   TextField "input_stall_1" at 225,144 size 180x20; Text 'MAN Manual'
   TextField "input_earth_1" at 225,168 size 180x20; Text 'SS Single Strt'
   TextField "input_ubal_1" at 225,192 size 180x20; Text 'TESTP Test Pem'
   TextField "Output_head_4" at 202,68 size 119x19; Text 'Output Modes'
   TextField "output_head_5" at 13,291 size 43x19; Text 'Reset'
   IOField "status_bit_1g_0r_16" at 72,96 size 20x20; FormatPattern 1; Unit  
      ProcessValue <- ".DQ.OK"
      Appearance <- ".DQ.OK"
   IOField "status_bit_1g_0r_17" at 72,120 size 20x20; FormatPattern 1; Unit  
      ProcessValue <- ".DQ.SACK"
      Appearance <- ".DQ.SACK"
   IOField "status_bit_1g_0r_18" at 72,144 size 20x20; FormatPattern 1; Unit  
      Appearance <- ".DQ.POS1"
      ProcessValue <- ".DQ.POS1"
   IOField "status_bit_1grn_0gry_6" at 72,168 size 20x20; FormatPattern 1; Unit  
      Appearance <- ".DQ.POS2"
      ProcessValue <- ".DQ.POS2"
   IOField "status_bit_1grn_0gry_7" at 72,192 size 20x20; FormatPattern 1; Unit  
      ProcessValue <- ".DQ.CON1"
      Appearance <- ".DQ.CON1"
   IOField "status_bit_1g_0r_22" at 276,92 size 20x20; FormatPattern 1; Unit  
      ProcessValue <- ".DQ.LOC"
      Appearance <- ".DQ.LOC"
   IOField "status_bit_1g_0r_23" at 276,120 size 20x20; FormatPattern 1; Unit  
      ProcessValue <- ".DQ.AUT"
      Appearance <- ".DQ.AUT"
   IOField "status_bit_1g_0r_24" at 276,144 size 20x20; FormatPattern 1; Unit  
      ProcessValue <- ".DQ.MAN"
      Appearance <- ".DQ.MAN"
   IOField "status_bit_1g_0r_25" at 276,168 size 20x20; FormatPattern 1; Unit  
      ProcessValue <- ".DQ.SS"
      Appearance <- ".DQ.SS"
   IOField "status_bit_1g_0r_26" at 276,192 size 20x20; FormatPattern 1; Unit  
      ProcessValue <- ".DQ.TESTP"
      Appearance <- ".DQ.TESTP"
   Button "btn_reset" at 172,318 size 80x30; TextOff 'Reset'
      on Click: SetBit(".FP_CMD.Reset")
      ObjectEnable <- ".FP_DIM.Reset"
      Visibility <- ".FP_SHOW.PB_Reset"
   TextField "output_con1_2" at 24,216 size 200x20; Text 'CON2 Cmd Close'
   IOField "status_bit_1grn_0gry_4" at 72,216 size 20x20; FormatPattern 1; Unit  
      ProcessValue <- ".DQ.CON2"
      Appearance <- ".DQ.CON2"
   TextField "output_con1_3" at 24,240 size 200x20; Text 'RES Reset'
   IOField "status_bit_1grn_0gry_5" at 72,240 size 20x20; FormatPattern 1; Unit  
      Appearance <- ".DQ.RES"
      ProcessValue <- ".DQ.RES"
   TextField "output_con1_4" at 24,263 size 200x20; Text 'ASTW Str Warn'
   IOField "status_bit_1grn_0gry_8" at 72,263 size 20x20; FormatPattern 1; Unit  
      ProcessValue <- ".DQ.CON1"
      Appearance <- ".DQ.ASTW"
   TextField "output_head_1" at 16,69 size 49x19; Text 'Timers'
   TextField "timers_text" at 24,96 size 100x20; Text 'Lim Drifting'
   IOField "delay_start_tm_sp" at 132,96 size 60x20; Authorization "User administration"; FormatPattern 9999; Unit  s
      ProcessValue <- ".FP_PARM.DriftingTime_Pre"
   TextField "timers_text_1" at 24,120 size 100x20; Text 'Run Time'
   TextField "timers_text_2" at 24,144 size 100x20; Text 'Delayed Start'
   TextField "timers_text_3" at 24,168 size 100x20; Text 'Delayed Stop'
   TextField "timers_text_4" at 24,192 size 100x20; Text 'Start Warning'
   IOField "return_tm_sp" at 132,120 size 60x20; Authorization "User administration"; FormatPattern 9999; Unit  s
      ProcessValue <- ".FP_PARM.RunTime_Pre"
   IOField "delayed_run_tm_sp" at 132,144 size 60x20; Authorization "User administration"; FormatPattern 9999; Unit  s
      ProcessValue <- ".FP_PARM.DelayStart_Pre"
   IOField "delay_stop_tm_sp" at 132,168 size 60x20; Authorization "User administration"; FormatPattern 999; Unit  s
      ProcessValue <- ".FP_PARM.DelayStop_Pre"
   IOField "delay_startsrm_tm_sp" at 132,192 size 60x20; Authorization "User administration"; FormatPattern 999; Unit  s
      ProcessValue <- ".FP_PARM.StartWarn_Pre"
   TextField "output_head_2" at 16,69 size 50x19; Text 'Spare'
   TextField "output_head_6" at 15,196 size 50x19; Text 'Spare'
   TextField "output_head_7" at 14,324 size 45x19; Text 'Spare'
   TextField "output_head_8" at 20,70 size 82x19; Text 'Supression'
   CheckBox "Check box_1" at 28,96 size 180x20; Text0 'Alarm Supression'; Authorization "User administration"
   TextField "output_head_14" at 16,68 size 103x19; Text 'Displat Inputs'
   CheckBox "cb_Type_Indication_1" at 16,100 size 100x20; Text0 'RDY'; Authorization "User administration"
      ProcessValue <- ".FP_SHOW.RDY"
   TextField "output_head_22" at 16,196 size 178x19; Text 'Relation to Group object'
   CheckBox "Check box_5" at 12,220 size 188x20; Text0 'Inherit Moded from Grp'; Authorization "User administration"
      ProcessValue <- ".FP_SEL.GroupMode"
   CheckBox "Check box_6" at 12,244 size 188x20; Text0 'Controled from Grp'; Authorization "User administration"
      ProcessValue <- ".FP_SEL.GroupCtrl"
   CheckBox "cb_Type_Indication_4" at 16,124 size 100x20; Text0 'OVL'; Authorization "User administration"
      ProcessValue <- ".FP_SHOW.OVL"
   CheckBox "cb_Type_Indication_5" at 16,148 size 100x20; Text0 'REM'; Authorization "User administration"
      ProcessValue <- ".FP_SHOW.REM"
   CheckBox "cb_Type_Indication_2" at 112,100 size 100x20; Text0 'SSW'; Authorization "User administration"
      ProcessValue <- ".FP_SHOW.SSW"
   CheckBox "cb_Type_Indication_6" at 112,124 size 100x20; Text0 'DRDY'; Authorization "User administration"
      ProcessValue <- ".FP_SHOW.DRDY"
   CheckBox "cb_Type_Indication_7" at 112,148 size 100x20; Text0 'GFA'; Authorization "User administration"
      ProcessValue <- ".FP_SHOW.GFA"
   CheckBox "cb_Type_Indication_8" at 204,100 size 100x20; Text0 'GWA'; Authorization "User administration"
      ProcessValue <- ".FP_SHOW.GWA"
   CheckBox "cb_Type_Indication_9" at 204,124 size 100x20; Text0 'BUSF'; Authorization "User administration"
      ProcessValue <- ".FP_SHOW.BUSF"
   CheckBox "cb_Type_Indication_10" at 204,148 size 100x20; Text0 'UTEST'; Authorization "User administration"
      ProcessValue <- ".FP_SHOW.UTEST"
   CheckBox "cb_Type_Indication_11" at 300,100 size 100x20; Text0 'RDY'; Authorization "User administration"
      ProcessValue <- ".FP_SHOW.RDY"
   CheckBox "cb_Type_Indication_12" at 300,124 size 100x20; Text0 'ACK'; Authorization "User administration"
      ProcessValue <- ".FP_SHOW.ACK"
   TextField "output_head_15" at 15,68 size 114x19; Text 'PLC Subroutine'
   TextField "text_16" at 24,92 size 100x20; Text 'SubRoutine'
   TextField "text_1" at 24,120 size 100x20; Text 'Version'
   IOField "iof_vers" at 136,120 size 60x20; FormatPattern 9999; Unit  
      ProcessValue <- "[0]"
   TextField "text_2" at 24,148 size 100x20; Text 'Build'
   IOField "iof_build" at 136,148 size 60x20; FormatPattern 9999; Unit  
      ProcessValue <- "[1]"
   TextField "text_3" at 24,176 size 100x20; Text 'IOSys'
   TextField "output_head_18" at 212,68 size 129x19; Text 'Program Status'
   TextField "text_4" at 226,92 size 100x20; Text 'State Pointer'
   IOField "iof_state_pointer" at 338,92 size 60x20; FormatPattern 9999; Unit  
      ProcessValue <- ".BlockInfo[2]"
   TextField "text_5" at 227,120 size 100x20; Text 'State Pointer_Prev'
   IOField "iof_state_pointer_prev" at 339,120 size 60x20; FormatPattern 9999; Unit  
      ProcessValue <- ".BlockInfo[3]"
   TextField "output_head_19" at 16,228 size 106x19; Text 'PLC Reference'
   TextField "text_6" at 24,256 size 100x20; Text 'DB'
   IOField "iof_db" at 136,256 size 60x20; FormatPattern 9999; Unit  
      ProcessValue <- ".BlockInfo[4]"
   TextField "output_head_20" at 16,292 size 51x19; Text 'EcsRef'
   TextField "output_head_21" at 16,412 size 79x19; Text 'ParentInfo'
   TextField "text_7" at 24,320 size 100x20; Text 'FP Name'
   TextField "text_8" at 24,348 size 100x20; Text 'Blk Alg Ver'
   TextField "text_9" at 24,376 size 100x20; Text 'Status Alg Ver'
   IOField "parent_info" at 24,440 size 380x20; FormatPattern *; Unit  
      ProcessValue <- ".ParentInfo"
   TextField "output_head_9" at 20,70 size 74x19; Text 'Unit Type'
   CheckBox "cb_Type_Indication" at 12,144 size 180x20; Text0 'Indication'; Authorization "User administration"
      ProcessValue <- ".FP_SEL.Type_Indication"
   OptionGroup "op_Type_Unimotor" at 12,96 size 180x20; Text0 '2 Pos Valve'; Authorization "User administration"
      ProcessValue <- ".FP_SEL.Type_2Pos"
   OptionGroup "op_Type_Bimotor" at 12,120 size 180x20; Text0 '3 Pos Valve'; Authorization "User administration"
      ProcessValue <- ".FP_SEL.Type_3Pos"
   CheckBox "cb_OutOfSevice" at 12,168 size 180x20; Text0 'Without Lim Switch'; Authorization "User administration"
      ProcessValue <- ".FP_SEL.Type_NoLimit"
   TextField "output_head_10" at 188,70 size 164x19; Text 'Start Warning Enable'
   CheckBox "cb_STW_Single" at 200,96 size 180x20; Text0 'Single Start'; Authorization "User administration"
      ProcessValue <- ".FP_SEL.STW_Single"
   CheckBox "cb_STW_Manual" at 200,120 size 180x20; Text0 'Manual'; Authorization "User administration"
      ProcessValue <- ".FP_SEL.STW_Manual"
   CheckBox "cb_STW_AutoStart" at 200,144 size 188x20; Text0 'Intrval Str (Auto Start)'; Authorization "User administration"
      ProcessValue <- ".FP_SEL.STW_AutoStart"
   CheckBox "cb_STW_Loca" at 200,168 size 188x20; Text0 'Local'; Authorization "User administration"
      ProcessValue <- ".FP_SEL.STW_Local"
   TextField "output_head_11" at 20,222 size 107x19; Text 'Alarm Handing'
   TextField "output_head_12" at 188,222 size 112x19; Text 'Enable Modes'
   CheckBox "Check box_8" at 12,248 size 180x20; Text0 'Warning Drive'; Authorization "User administration"
      ProcessValue <- ".FP_SEL.WarningDrive"
   CheckBox "Check box_9" at 12,272 size 180x20; Text0 'Sup by Parent Grp'; Authorization "User administration"
      ProcessValue <- ".FP_SEL.ParentSupress"
   CheckBox "Check box_10" at 12,296 size 188x20; Text0 'Pass Status to Par Grp'; Authorization "User administration"
      ProcessValue <- ".FP_SEL.ParentCollection"
   CheckBox "Check box_11" at 200,248 size 180x20; Text0 'Automatic'; Authorization "User administration"
      ProcessValue <- ".FP_EN.Mode_Auto"
   CheckBox "Check box_12" at 200,272 size 180x20; Text0 'Manual'; Authorization "User administration"
      ProcessValue <- ".FP_EN.Mode_Man"
   CheckBox "Check box_13" at 200,296 size 188x20; Text0 'Local'; Authorization "User administration"
      ProcessValue <- ".FP_EN.Mode_Loc"
   CheckBox "Check box_14" at 200,320 size 188x20; Text0 'Single Start FP'; Authorization "User administration"
      ProcessValue <- ".FP_EN.Mode_SS_FP"
   CheckBox "Check box_15" at 200,344 size 188x20; Text0 'Single Start Filed'; Authorization "User administration"
      ProcessValue <- ".FP_EN.Mode_SS_Field"
   CheckBox "Check box_16" at 200,368 size 188x20; Text0 'Test mode'; Authorization "User administration"
      ProcessValue <- ".FP_EN.Mode_Test"
   TextField "output_head_13" at 20,393 size 116x19; Text 'Enable Features'
   CheckBox "Check box_19" at 12,416 size 188x20; Text0 'Quick Stop frm Unit'; Authorization "User administration"
      ProcessValue <- ".FP_EN.PB_QStop"
   CheckBox "Check box_20" at 12,440 size 188x20; Text0 'Reset Btn on FP'; Authorization "User administration"
      ProcessValue <- ".FP_SHOW.PB_Reset"
   TextField "output_head_16" at 188,391 size 187x19; Text 'Park Pos when Grp Stop'
   CheckBox "cb_OutOfSevice_1" at 12,192 size 180x20; Text0 'Out of Sevices'; Authorization "User administration"
      ProcessValue <- ".FP_SEL.OutOfSevice"
   TextField "output_head_17" at 20,320 size 127x19; Text 'Output Cmd Type'
   OptionGroup "op_Type_Unimotor_1" at 12,344 size 180x20; Text0 'Constant'; Authorization "User administration"
      ProcessValue <- ".FP_SEL.Type_ConstantCmd"
   OptionGroup "op_Type_Bimotor_1" at 12,368 size 180x20; Text0 'Pulse'; Authorization "User administration"
      ProcessValue <- ".FP_SEL.Type_PulseCmd"
   CheckBox "Check box_2" at 200,416 size 188x20; Text0 'Current Pos'; Authorization "User administration"
      ProcessValue <- ".FP_SEL.Park_CurrPos"
   CheckBox "Check box_3" at 200,440 size 188x20; Text0 'Open Pos'; Authorization "User administration"
      ProcessValue <- ".FP_SEL.Park_Pos1"
   CheckBox "Check box_4" at 200,464 size 188x20; Text0 'Close Pos'; Authorization "User administration"
      ProcessValue <- ".FP_SEL.Park_Pos2"
   TextField "interlockl_head_1" at 16,68 size 99x22; Text 'Interlocking'
   TextField "interlockl_head_2" at 16,379 size 180x22; Text 'Sequence Interlocking'
   TextField "interlockl_head_3" at 16,192 size 158x22; Text 'Sequence Int Open'
   TextField "interlock_1" at 24,100 size 140x20; Text 'Interlock 1'
      Text <- ".INTL01.DefaultText"
      Visibility <- ".INTL01"
   TextField "interlock_2" at 24,128 size 140x20; Text 'Interlock 2'
      Text <- ".INTL02.DefaultText"
      Visibility <- ".INTL04"
   TextField "interlock_3" at 24,156 size 140x20; Text 'Interlock 3'
      Text <- ".INTL03.DefaultText"
      Visibility <- ".INTL04"
   TextField "STRT_1" at 24,407 size 140x20; Text 'Interlock 1'
      Text <- ".INTL_SEQ_STP01.DefaultText"
      Visibility <- ".INTL_SEQ_STP01"
   TextField "STRT_2" at 24,435 size 140x20; Text 'Interlock 2'
      Visibility <- ".INTL_SEQ_STP02"
      Text <- ".INTL_SEQ_STP02.DefaultText"
   TextField "STRT_3" at 216,408 size 140x20; Text 'Interlock 3'
      Text <- ".INTL_SEQ_STP03.DefaultText"
      Visibility <- ".INTL_SEQ_STP03"
   TextField "STRT_4" at 216,436 size 140x20; Text 'Interlock 4'
      Visibility <- ".INTL_SEQ_STP04"
      Text <- ".INTL_SEQ_STP04.DefaultText"
   SymbolicIOField "int_01" at 160,100 size 45x20; TextOn '1'; TextOff '0'; TextList "interlock_status_byte"
      Appearance <- ".INTL01"
      ProcessValue <- ".INTL01"
      Visibility <- ".INTL01"
   SymbolicIOField "int_2" at 160,128 size 45x20; TextOn '1'; TextOff '0'; TextList "interlock_status_byte"
      Visibility <- ".INTL02"
      ProcessValue <- ".INTL02"
      Appearance <- ".INTL02"
   SymbolicIOField "int_1" at 160,156 size 45x20; TextOn '1'; TextOff '0'; TextList "interlock_status_byte"
      Visibility <- ".INTL03"
      ProcessValue <- ".INTL03"
      Appearance <- ".INTL03"
   TextField "interlock_5" at 221,100 size 140x20; Text 'Interlock 4'
      Text <- ".INTL04.DefaultText"
      Visibility <- ".INTL04"
   TextField "interlock_6" at 221,128 size 140x20; Text 'Interlock 5'
      Text <- ".INTL05.DefaultText"
      Visibility <- ".INTL05"
   TextField "interlock_7" at 221,156 size 140x20; Text 'Interlock 6'
      Text <- ".INTL07.DefaultText"
      Visibility <- ".INTL06"
   SymbolicIOField "int_4" at 357,100 size 45x20; TextOn '1'; TextOff '0'; TextList "interlock_status_byte"
      ProcessValue <- ".INTL04"
      Visibility <- ".INTL04"
      Appearance <- ".INTL04"
   SymbolicIOField "int_5" at 357,128 size 45x20; TextOn '1'; TextOff '0'; TextList "interlock_status_byte"
      Appearance <- ".INTL04"
      Visibility <- ".INTL04"
      ProcessValue <- ".INTL04"
   SymbolicIOField "int_6" at 356,156 size 45x20; TextOn '1'; TextOff '0'; TextList "interlock_status_byte"
      Visibility <- ".INTL06"
      Appearance <- ".INTL06"
      ProcessValue <- ".INTL06"
   SymbolicIOField "int_8" at 160,407 size 45x20; TextOn '1'; TextOff '0'; TextList "interlock_status_byte"
      Visibility <- ".INTL_SEQ_STP01"
      Appearance <- ".INTL_SEQ_STP01"
      ProcessValue <- ".INTL_SEQ_STP01"
   SymbolicIOField "int_9" at 160,435 size 45x20; TextOn '1'; TextOff '0'; TextList "interlock_status_byte"
      Visibility <- ".INTL_SEQ_STP02"
      Appearance <- ".INTL_SEQ_STP02"
      ProcessValue <- ".INTL_SEQ_STP02"
   SymbolicIOField "int_10" at 352,408 size 45x20; TextOn '1'; TextOff '0'; TextList "interlock_status_byte"
      Visibility <- ".INTL_SEQ_STP03"
      Appearance <- ".INTL_SEQ_STP03"
      ProcessValue <- ".INTL_SEQ_STP03"
   SymbolicIOField "int_11" at 352,436 size 45x20; TextOn '1'; TextOff '0'; TextList "interlock_status_byte"
      Visibility <- ".INTL_SEQ_STP04"
      Appearance <- ".INTL_SEQ_STP04"
      ProcessValue <- ".INTL_SEQ_STP04"
   TextField "STP_1" at 24,221 size 140x20; Text 'Interlock 1'
      Visibility <- ".INTL_SEQ_STR1_01"
      Text <- ".INTL_SEQ_STR1_01.DefaultText"
   TextField "STP_2" at 24,249 size 140x20; Text 'Interlock 2'
      Text <- "..INTL_SEQ_STR1_02.DefaultText"
      Visibility <- ".INTL_SEQ_STR1_02"
   TextField "STP_3" at 220,220 size 140x20; Text 'Interlock 3'
      Text <- ".INTL_SEQ_STR1_03.DefaultText"
      Visibility <- ".INTL_SEQ_STR1_03"
   SymbolicIOField "stp_int_1" at 160,221 size 45x20; TextOn '1'; TextOff '0'; TextList "interlock_status_byte"
      ProcessValue <- ".INTL_SEQ_STR1_01"
      Visibility <- ".INTL_SEQ_STR1_01"
      Appearance <- ".INTL_SEQ_STR1_01"
   SymbolicIOField "stp_int_2" at 160,249 size 45x20; TextOn '1'; TextOff '0'; TextList "interlock_status_byte"
      Visibility <- ".INTL_SEQ_STR1_02"
      Appearance <- ".INTL_SEQ_STR1_02"
      ProcessValue <- ".INTL_SEQ_STR1_02"
   SymbolicIOField "stp_int_3" at 356,220 size 45x20; TextOn '1'; TextOff '0'; TextList "interlock_status_byte"
      Visibility <- ".INTL_SEQ_STR1_03"
      Appearance <- ".INTL_SEQ_STR1_03"
      ProcessValue <- ".INTL_SEQ_STR1_03"
   TextField "STP_4" at 220,248 size 140x20; Text 'Interlock 4'
      Visibility <- ".INTL_SEQ_STR1_04"
      Text <- "..INTL_SEQ_STR1_04.DefaultText"
   SymbolicIOField "stp_int_4" at 356,248 size 45x20; TextOn '1'; TextOff '0'; TextList "interlock_status_byte"
      Visibility <- ".INTL_SEQ_STR1_04"
      Appearance <- ".INTL_SEQ_STR1_04"
      ProcessValue <- ".INTL_SEQ_STR1_04"
   TextField "interlockl_head_4" at 16,288 size 158x22; Text 'Sequence Int Close'
   TextField "STP_5" at 24,313 size 140x20; Text 'Interlock 1'
      Visibility <- ".INTL_SEQ_STR2_01"
      Text <- ".INTL_SEQ_STR2_01.DefaultText"
   TextField "STP_6" at 24,341 size 140x20; Text 'Interlock 2'
      Visibility <- ".INTL_SEQ_STR2_02"
      Text <- "..INTL_SEQ_STR2_02.DefaultText"
   TextField "STP_7" at 220,312 size 140x20; Text 'Interlock 3'
      Visibility <- ".INTL_SEQ_STR2_03"
      Text <- ".INTL_SEQ_STR2_03.DefaultText"
   SymbolicIOField "stp_int_5" at 160,313 size 45x20; TextOn '1'; TextOff '0'; TextList "interlock_status_byte"
      Visibility <- ".INTL_SEQ_STR2_01"
      Appearance <- ".INTL_SEQ_STR2_01"
      ProcessValue <- ".INTL_SEQ_STR2_01"
   SymbolicIOField "stp_int_6" at 160,341 size 45x20; TextOn '1'; TextOff '0'; TextList "interlock_status_byte"
      Visibility <- ".INTL_SEQ_STR2_02"
      Appearance <- ".INTL_SEQ_STR2_02"
      ProcessValue <- ".INTL_SEQ_STR2_02"
   SymbolicIOField "stp_int_7" at 356,312 size 45x20; TextOn '1'; TextOff '0'; TextList "interlock_status_byte"
      Visibility <- ".INTL_SEQ_STR2_03"
      Appearance <- ".INTL_SEQ_STR2_03"
      ProcessValue <- ".INTL_SEQ_STR2_03"
   TextField "STP_8" at 220,340 size 140x20; Text 'Interlock 4'
      Text <- "..INTL_SEQ_STR2_04.DefaultText"
      Visibility <- ".INTL_SEQ_STR2_04"
   SymbolicIOField "stp_int_8" at 356,340 size 45x20; TextOn '1'; TextOff '0'; TextList "interlock_status_byte"
      Visibility <- ".INTL_SEQ_STR2_04"
      Appearance <- ".INTL_SEQ_STR2_04"
      ProcessValue <- ".INTL_SEQ_STR2_04"

screen "Main" 1280x728
   ScreenModuleView "motor_3" at 84,124 size 115x71; Guid_{11997190-12899} 'G21'; Guid_{11997190-11745} '020PU043U01'; Guid_{11997190-13883} 'Насосы отопления'; ScreenModuleType ""
      Guid_{11997190-10442} <- "020PU043U01.MSW"
      on ReleaseLeft: "OnReleaseLeft"
   ScreenModuleView "valve_2" at 204,324 size 115x67; Guid_{11997190-11745} '2080SP241Y01'; ScreenModuleType ""
      on ReleaseLeft: "OnReleaseLeft"
      Guid_{11997190-10442} <- "2080SP241Y01.MSW"
   Button "Button_4" at 1184,680 size 80x30; TextOff 'Logon'
      on Click: function_a2a04561()
   TextField "Text field_3" at 1116,656 size 150x21; Text 'User'
      Text <- "@CurrentUser"
   TextField "Text field_6" at 1136,588 size 131x59; Text 'Admin:admin1 Operator:operator Viwer:viwer1'
   Button "Button_1" at 1120,352 size 80x30; TextOff 'Text'; Authorization "Operate"
      on Click: "OnClick"
      on ReleaseLeft: "OnReleaseLeft"
   ScreenModuleView "motor_1" at 84,212 size 115x71; Guid_{11997190-12899} 'G21'; Guid_{11997190-11745} '020PU044U01'; Guid_{11997190-13883} 'Насосы отопления'; ScreenModuleType ""
      on ReleaseLeft: "OnReleaseLeft"
      Guid_{11997190-10442} <- "020PU044U01.MSW"
   ScreenModuleView "motor_2" at 84,320 size 115x71; Guid_{11997190-12899} 'G21'; Guid_{11997190-11745} '2080SP241U01'; Guid_{11997190-13883} 'Насосы отопления'; ScreenModuleType ""
      on ReleaseLeft: "OnReleaseLeft"
      Guid_{11997190-10442} <- "2080SP241U01.MSW"
   ScreenModuleView "analog_1" at 208,132 size 134x47; Guid_{11997190-11745} '2080SP241U01S01'; ScreenModuleType ""
      Guid_{11997190-10442} <- "2080SP241U01S01.MSW"
      Guid_{11997190-34420} <- "2080SP241U01S01.Unit"
      on ReleaseLeft: "OnReleaseLeft"
      Guid_{11997190-36353} <- "2080SP241U01S01.Decimals"
      Guid_{11997191-34289} <- "VALUE"
      Guid_{11997191-34295} <- "EXT"
      Guid_{11997191-34297} <- "Status"
   ScreenModuleView "analog_3" at 1120,36 size 134x47; Guid_{11997190-11745} '2080TN450A01F01'; ScreenModuleType ""
      on ReleaseLeft: "OnReleaseLeft"
      Guid_{11997190-10442} <- "2080TN450A01F01.MSW"
      Guid_{11997190-34420} <- "2080TN450A01F01.Unit"
      Guid_{11997190-36353} <- "2080TN450A01F01.Decimals"
      Guid_{11997191-34289} <- "VALUE"
      Guid_{11997191-34295} <- "EXT"
      Guid_{11997191-34297} <- "Status"
   ScreenModuleView "analog_4" at 208,164 size 134x47; Guid_{11997190-11745} '2080TN450A01I02'; ScreenModuleType ""
      on ReleaseLeft: "OnReleaseLeft"
      Guid_{11997190-10442} <- "2080TN450A01I02.MSW"
      Guid_{11997190-34420} <- "2080TN450A01I02.Unit"
      Guid_{11997190-36353} <- "2080TN450A01I02.Decimals"
      Guid_{11997191-34289} <- "VALUE"
      Guid_{11997191-34295} <- "EXT"
      Guid_{11997191-34297} <- "Status"
   ScreenModuleView "motor_4" at 84,412 size 115x71; Guid_{11997190-12899} 'G21'; Guid_{11997190-11745} '2080SP242U01'; Guid_{11997190-13883} 'Насосы отопления'; ScreenModuleType ""
      on ReleaseLeft: "OnReleaseLeft"
      Guid_{11997190-10442} <- "2080SP242U01.MSW"
   ScreenModuleView "valve_1" at 204,416 size 115x67; Guid_{11997190-11745} '2080SP242Y01'; ScreenModuleType ""
      on ReleaseLeft: "OnReleaseLeft"
      Guid_{11997190-10442} <- "2080SP242Y01.MSW"
   ScreenModuleView "analog_5" at 208,196 size 134x47; Guid_{11997190-11745} '2910RS001A01N01'; ScreenModuleType ""
      on ReleaseLeft: "OnReleaseLeft"
      Guid_{11997190-10442} <- "2910RS001A01N01.MSW"
      Guid_{11997190-34420} <- "2910RS001A01N01.Unit"
      Guid_{11997190-36353} <- "2910RS001A01N01.Decimals"
      Guid_{11997191-34289} <- "VALUE"
      Guid_{11997191-34295} <- "EXT"
      Guid_{11997191-34297} <- "Status"
   ScreenModuleView "analog_6" at 1120,108 size 134x47; Guid_{11997190-11745} '2910RS001A01L02'; ScreenModuleType ""
      on ReleaseLeft: "OnReleaseLeft"
      Guid_{11997190-36353} <- "2910RS001A01L02.Decimals"
      Guid_{11997190-10442} <- "2910RS001A01L02.MSW"
      Guid_{11997190-34420} <- "2910RS001A01L02.Unit"
      Guid_{11997191-34289} <- "VALUE"
      Guid_{11997191-34295} <- "EXT"
      Guid_{11997191-34297} <- "Status"
   Button "Button_2" at 1120,252 size 80x30; TextOff 'Text'
      on ReleaseLeft: function_c00bc162("Main", "w_popup_unit_1", ScreenName, 'fp_valve'); function_c00bc162("Main", "w_popup_unit_1", TagPrefix, '2080SP241Y01'); function_c00bc162("Main", "w_popup_unit_1", Visible, 'true')
   Button "Button_3" at 1120,292 size 80x30; TextOff 'Text'
      on ReleaseLeft: "OnReleaseLeft"
   ScreenModuleView "motor_5" at 84,620 size 115x71; Guid_{11997190-12899} 'G21'; Guid_{11997190-11745} '2080SP242U01'; Guid_{11997190-13883} 'Насосы отопления'; ScreenModuleType ""
      Guid_{11997190-10442} <- "2080SP242U01.MSW"
      on ReleaseLeft: "OnReleaseLeft"
   ScreenWindow "w_popup_unit_1" at 100,24 size 520x540; CaptionText 'UNIT'; ScreenName "fp_motor"
   ScreenWindow "w_popup_unit_2" at 112,56 size 520x540; CaptionText 'UNIT'
   ScreenWindow "w_popup_unit_3" at 124,84 size 520x540; CaptionText 'UNIT'
   ScreenWindow "w_popup_unit_4" at 136,116 size 520x540; CaptionText 'UNIT'
   ScreenWindow "w_popup_unit_5" at 148,148 size 520x540; CaptionText 'UNIT'
   TextField "Text field_1" at 41,24 size 136x25; Text 'Не удалять!'
   TextField "ord_ppopup_win" at 341,44 size 16x32; ToolTipText 'След window в которое будет загружен попап screen'; Text '0'
   TextField "Text field_2" at 41,56 size 288x18; Text 'Номер очереди popup ScreenWindow:'

screen "fp_analog" 500x500
   on GenerateScreen: "show_tab"(1)
   TextField "cntrl_box_cntrl_head" at 12,100 size 60x22; Text 'Analog'
   Bar "Bar_1" at 136,128 size 144x352; MinimumValue 0; MaximumValue 100
      MaximumValue <- ".FP_PARAM.Scale_Max"
      MinimumValue <- ".FP_PARAM.Scale_Min"
      ProcessValue <- ".MSW.VALUE"
      Unit <- ".Unit"
      AlarmUpperLimit <- ".FP_PARAM.AlarmLimit_H3"
      AlarmLowerLimit <- ".FP_PARAM.AlarmLimit_L3"
      WarningUpperLimit <- ".FP_PARAM.AlarmLimit_H2"
      WarningLowerLimit <- ".FP_PARAM.AlarmLimit_L2"
      AlarmUpperLimitEnabled <- ".FP_EN.Alarm_H3"
      WarningUpperLimitEnabled <- ".FP_EN.Alarm_H2"
      AlarmLowerLimitEnabled <- ".FP_EN.Alarm_L3"
      WarningLowerLimitEnabled <- ".FP_EN.Alarm_L2"
   TextField "header_txt" at 8,8 size 396x21; Text 'HEADER'
      Text <- ".DefaultText"
   SymbolicIOField "status I/O field_1" at 8,32 size 396x32; TextOn '1'; TextOff '0'; TextList "analog_status"
      ProcessValue <- ".StatusWork"
      Appearance <- ".StatusWork"
   Button "bt_tab_1" at 412,109 size 80x28; TextOff 'Main'
      on Click: "show_tab"(1)
   Button "bt_tab_3" at 412,172 size 80x28; TextOff 'Input'
      on Click: "show_tab"(3)
   Button "bt_tab_4" at 412,204 size 80x28; TextOff 'Output'
      on Click: "show_tab"(4)
   Button "bt_tab_5" at 412,236 size 80x28; TextOff 'Limits'
      on Click: "show_tab"(5)
   Button "bt_tab_6" at 412,268 size 80x28; TextOff 'Scale'
      on Click: "show_tab"(6)
   Button "bt_tab_7" at 412,300 size 80x28; TextOff 'Point para'
      on Click: "show_tab"(7)
   Button "bt_tab_8" at 412,332 size 80x28; TextOff 'Config'
      on Click: "show_tab"(8)
   Button "bt_tab_11" at 412,396 size 80x28; TextOff 'Info'
      on Click: "show_tab"(11)
   Button "bt_tab_9" at 412,364 size 80x28; TextOff 'Treat'
      on Click: "show_tab"(9)
   Button "bt_tab_2" at 412,141 size 80x28; TextOff 'Trend'
      on Click: "show_tab"(2)
   IOField "I/O value" at 4,71 size 400x20; FormatPattern s99999.999
      ProcessValue <- ".MSW.VALUE"
      Unit <- ".Unit"
      FormatPattern <- ".Decimals"
      Appearance <- ".StatusWork"
   TextField "output_head_25" at 13,37 size 22x22; Text '!'
      Visibility <- ".FP_EN.Force"
   TextField "input_head" at 15,100 size 38x19; Text 'Input'
   TextField "input_rdy" at 20,204 size 200x20; Text 'U_RANGE Under Range'
   TextField "input_mcc" at 20,228 size 200x20; Text 'O_RANGE Over Range'
   TextField "input_ovl" at 20,252 size 200x20; Text 'SIG_FAULT SIG_FAULT'
   TextField "input_ret1" at 20,276 size 200x20; Text 'EnConfig EnConfig'
   TextField "input_lstr1" at 20,300 size 200x20; Text 'AEN Alarm Enable'
   TextField "input_lstp" at 20,324 size 200x20; Text 'AL_SUPR Alarm Suppress'
   IOField "status_bit_1g_0r_3" at 88,204 size 20x20; FormatPattern 1; Unit  
      ProcessValue <- ".DI.U_RANGE"
      Appearance <- ".DI.U_RANGE"
   IOField "status_bit_1g_0r_2" at 88,228 size 20x20; FormatPattern 1; Unit  
      ProcessValue <- ".DI.O_RANGE"
      Appearance <- ".DI.O_RANGE"
   IOField "status_bit_1g_0r_4" at 88,252 size 20x20; FormatPattern 1; Unit  
      ProcessValue <- ".DI.SIG_FAULT"
      Appearance <- ".DI.SIG_FAULT"
   IOField "status_bit_1grn_0gry_5" at 88,276 size 20x20; FormatPattern 1; Unit  
      Appearance <- ".DI.RET1"
      ProcessValue <- ".DI.EnConfig"
   IOField "status_bit_1grn_0gry_1" at 88,300 size 20x20; FormatPattern 1; Unit  
      ProcessValue <- ".DI.AEN"
      Appearance <- ".DI.AEN"
   IOField "status_bit_1g_0r_5" at 88,324 size 20x20; FormatPattern 1; Unit  
      ProcessValue <- ".DI.AL_SUPR"
      Appearance <- ".DI.AL_SUPR"
   TextField "input_rdy_1" at 20,124 size 36x20; Text 'IN'
   IOField "status_bit_1g_0r_32" at 148,124 size 60x20; FormatPattern s999.9; Unit  
      ProcessValue <- ".I.IN"
   TextField "input_rdy_2" at 20,148 size 80x20; Text 'SIG TYPE'
   IOField "status_bit_1g_0r_33" at 148,148 size 60x20; FormatPattern 99; Unit  
      ProcessValue <- ".I.SIG_TYPE"
   TextField "input_rdy_3" at 20,172 size 120x20; Text 'FiledBus Status'
   IOField "status_bit_1g_0r_34" at 148,172 size 60x20; FormatPattern 999; Unit  
      ProcessValue <- ".I.FI_BUS"
   TextField "output_head_3" at 14,99 size 49x19; Text 'Output'
   TextField "input_rdy_4" at 20,176 size 200x20; Text 'AL_H3 H3 Fatal Alarm'
   TextField "input_mcc_1" at 20,200 size 200x20; Text 'AL_H2 H2 Alarm'
   TextField "input_ovl_1" at 20,224 size 200x20; Text 'AL_H1 H1 Warning'
   TextField "input_ret1_1" at 20,248 size 200x20; Text 'AL_L1 L1 Warning'
   TextField "input_lstr1_1" at 20,272 size 200x20; Text 'AL_L2 L2 Alarm'
   TextField "input_lstp_1" at 20,296 size 200x20; Text 'AL_L3 L3 Fatal Alarm'
   IOField "status_bit_1g_0r_1" at 88,176 size 20x20; FormatPattern 1; Unit  
      ProcessValue <- ".DQ.AL_H3"
      Appearance <- ".DQ.AL_H3"
   IOField "status_bit_1g_0r_6" at 88,200 size 20x20; FormatPattern 1; Unit  
      ProcessValue <- ".DQ.AL_H2"
      Appearance <- ".DQ.AL_H2"
   IOField "status_bit_1g_0r_7" at 88,224 size 20x20; FormatPattern 1; Unit  
      ProcessValue <- ".DQ.AL_H1"
      Appearance <- ".DQ.AL_H1"
   IOField "status_bit_1grn_0gry_2" at 88,248 size 20x20; FormatPattern 1; Unit  
      ProcessValue <- ".DQ.AL_L1"
      Appearance <- ".DQ.AL_L1"
   IOField "status_bit_1grn_0gry_3" at 88,272 size 20x20; FormatPattern 1; Unit  
      ProcessValue <- ".DQ.AL_L2"
      Appearance <- ".DQ.AL_L2"
   IOField "status_bit_1g_0r_8" at 88,296 size 20x20; FormatPattern 1; Unit  
      ProcessValue <- ".DQ.AL_L3"
      Appearance <- ".DQ.AL_L3"
   TextField "input_rdy_5" at 20,124 size 120x20; Text 'PV_NORM'
   IOField "status_bit_1g_0r_9" at 127,124 size 80x20; FormatPattern s999.9; Unit  
      ProcessValue <- ".Q.PV_NORM"
   TextField "input_rdy_6" at 20,148 size 120x20; Text 'PV_SCAL'
   IOField "status_bit_1g_0r_10" at 127,148 size 80x20; FormatPattern s999999999.9; Unit  
      ProcessValue <- ".Q.PV_SCAL"
      Unit <- ".Unit"
      FormatPattern <- ".Decimals"
   TextField "input_rdy_7" at 20,320 size 200x20; Text 'SIG_OK Signal OK'
   TextField "input_mcc_2" at 20,344 size 200x20; Text 'LIM_H2 Limit H2'
   TextField "input_ovl_2" at 20,368 size 200x20; Text 'LIM_H1 Limit H1'
   TextField "input_ret1_2" at 20,392 size 200x20; Text 'LIM_L1 Limit L1'
   TextField "input_lstr1_2" at 20,416 size 200x20; Text 'LIM_L2 Limit L2'
   TextField "input_lstp_2" at 20,440 size 200x20; Text 'GR_P Positive Limit'
   IOField "status_bit_1g_0r_11" at 88,320 size 20x20; FormatPattern 1; Unit  
      ProcessValue <- ".DQ.SIG_OK"
      Appearance <- ".DQ.SIG_OK"
   IOField "status_bit_1g_0r_12" at 88,344 size 20x20; FormatPattern 1; Unit  
      ProcessValue <- ".DQ.LIM_H2"
      Appearance <- ".DQ.LIM_H2"
   IOField "status_bit_1g_0r_13" at 88,368 size 20x20; FormatPattern 1; Unit  
      ProcessValue <- ".DQ.LIM_H1"
      Appearance <- ".DQ.LIM_H1"
   IOField "status_bit_1grn_0gry_4" at 88,392 size 20x20; FormatPattern 1; Unit  
      ProcessValue <- ".DQ.LIM_L1"
      Appearance <- ".DQ.LIM_L1"
   IOField "status_bit_1grn_0gry_6" at 88,416 size 20x20; FormatPattern 1; Unit  
      ProcessValue <- ".DQ.LIM_L2"
      Appearance <- ".DQ.LIM_L2"
   IOField "status_bit_1g_0r_14" at 88,440 size 20x20; FormatPattern 1; Unit  
      ProcessValue <- ".DQ.GR_P"
      Appearance <- ".DQ.GR_P"
   TextField "input_lstp_3" at 20,464 size 200x20; Text 'GR_N Negative Limit'
   IOField "status_bit_1g_0r_15" at 88,464 size 20x20; FormatPattern 1; Unit  
      ProcessValue <- ".DQ.GR_N"
      Appearance <- ".DQ.GR_N"
   TextField "output_head_1" at 9,102 size 90x19; Text 'Alarm Limits'
   IOField "delay_start_tm_sp" at 179,128 size 60x20; Authorization "User administration"; FormatPattern 9999
      ProcessValue <- ".FP_PARAM.AlarmLimit_H3"
      Unit <- ".Unit"
   IOField "return_tm_sp" at 179,152 size 60x20; Authorization "User administration"; FormatPattern 9999
      ProcessValue <- ".FP_PARAM.AlarmLimit_H2"
      Unit <- ".Unit"
   IOField "delayed_run_tm_sp" at 179,176 size 60x20; Authorization "User administration"; FormatPattern 9999
      ProcessValue <- ".FP_PARAM.AlarmLimit_H1"
      Unit <- ".Unit"
   IOField "delay_stop_tm_sp" at 179,200 size 60x20; Authorization "User administration"; FormatPattern 999
      ProcessValue <- ".FP_PARAM.AlarmLimit_L1"
      Unit <- ".Unit"
   IOField "delay_startsrm_tm_sp" at 179,224 size 60x20; Authorization "User administration"; FormatPattern 999
      ProcessValue <- ".FP_PARAM.AlarmLimit_L2"
      Unit <- ".Unit"
   TextField "output_head_22" at 248,102 size 102x19; Text 'Alarm Delay'
   IOField "delay_startsrm_tm_sp_1" at 179,248 size 60x20; Authorization "User administration"; FormatPattern 999
      ProcessValue <- ".FP_PARAM.AlarmLimit_L3"
      Unit <- ".Unit"
   CheckBox "Check box_2" at 4,128 size 188x20; Text0 'H3 Fatal Alarm'; Authorization "User administration"
      ProcessValue <- ".FP_EN.Alarm_H3"
   CheckBox "Check box_3" at 4,152 size 188x20; Text0 'H2 Alarm'; Authorization "User administration"
      ProcessValue <- ".FP_EN.Alarm_H2"
   CheckBox "Check box_4" at 4,176 size 188x20; Text0 'H1Warning'; Authorization "User administration"
      ProcessValue <- ".FP_EN.Alarm_H1"
   CheckBox "Check box_5" at 4,248 size 188x20; Text0 'L3 Fatal Alarm'; Authorization "User administration"
      ProcessValue <- ".FP_EN.Alarm_L3"
   CheckBox "Check box_6" at 4,224 size 188x20; Text0 'L2 Alarm'; Authorization "User administration"
      ProcessValue <- ".FP_EN.Alarm_L2"
   CheckBox "Check box_7" at 4,200 size 188x20; Text0 'L1Warning'; Authorization "User administration"
      ProcessValue <- ".FP_EN.Alarm_L1"
   IOField "delay_start_tm_sp_1" at 304,128 size 60x20; Authorization "User administration"; FormatPattern 9999; Unit  c
      ProcessValue <- ".FP_PARAM.AlarmDelay_H3_Pre"
   IOField "return_tm_sp_1" at 304,152 size 60x20; Authorization "User administration"; FormatPattern 9999; Unit  c
      ProcessValue <- ".FP_PARAM.AlarmDelay_H2_Pre"
   IOField "delayed_run_tm_sp_1" at 304,176 size 60x20; Authorization "User administration"; FormatPattern 9999; Unit  c
      ProcessValue <- ".FP_PARAM.AlarmDelay_H1_Pre"
   IOField "delay_stop_tm_sp_1" at 304,200 size 60x20; Authorization "User administration"; FormatPattern 999; Unit  c
      ProcessValue <- ".FP_PARAM.AlarmDelay_L1_Pre"
   IOField "delay_startsrm_tm_sp_2" at 304,224 size 60x20; Authorization "User administration"; FormatPattern 999; Unit  c
      ProcessValue <- ".FP_PARAM.AlarmDelay_L2_Pre"
   IOField "delay_startsrm_tm_sp_3" at 304,248 size 60x20; Authorization "User administration"; FormatPattern 999; Unit  c
      ProcessValue <- ".FP_PARAM.AlarmDelay_L3_Pre"
   CheckBox "Check box_27" at 264,128 size 32x20; Text0 'Text1'; Authorization "User administration"
      ProcessValue <- ".FP_EN.AlarmDelay_H3"
   CheckBox "Check box_28" at 264,152 size 32x20; Text0 'Text1'; Authorization "User administration"
      ProcessValue <- ".FP_EN.AlarmDelay_H2"
   CheckBox "Check box_29" at 264,176 size 32x20; Text0 'Text1'; Authorization "User administration"
      ProcessValue <- ".FP_EN.AlarmDelay_H1"
   CheckBox "Check box_30" at 264,248 size 32x20; Text0 'Text1'; Authorization "User administration"
      ProcessValue <- ".FP_EN.AlarmDelay_L3"
   CheckBox "Check box_31" at 264,224 size 32x20; Text0 'Text1'; Authorization "User administration"
      ProcessValue <- ".FP_EN.AlarmDelay_L2"
   CheckBox "Check box_32" at 264,200 size 32x20; Text0 'Text1'; Authorization "User administration"
      ProcessValue <- ".FP_EN.AlarmDelay_L1"
   IOField "status_bit_1g_0r_19" at 156,128 size 20x20; FormatPattern 1; Unit  
      ProcessValue <- ".DQ.AL_H3"
      Appearance <- ".DQ.AL_H3"
   IOField "status_bit_1g_0r_20" at 156,152 size 20x20; FormatPattern 1; Unit  
      Appearance <- ".DQ.AL_H2"
      ProcessValue <- ".DQ.AL_H2"
   IOField "status_bit_1g_0r_21" at 156,176 size 20x20; FormatPattern 1; Unit  
      ProcessValue <- ".DQ.AL_H1"
      Appearance <- ".DQ.AL_H1"
   IOField "status_bit_1g_0r_29" at 156,200 size 20x20; FormatPattern 1; Unit  
      Appearance <- ".DQ.AL_L1"
      ProcessValue <- ".DQ.AL_L1"
   IOField "status_bit_1g_0r_30" at 156,224 size 20x20; FormatPattern 1; Unit  
      ProcessValue <- ".DQ.AL_L2"
      Appearance <- ".DQ.AL_L2"
   IOField "status_bit_1g_0r_31" at 156,248 size 20x20; FormatPattern 1; Unit  
      Appearance <- ".DQ.AL_L3"
      ProcessValue <- ".DQ.AL_L3"
   TextField "output_head_23" at 9,292 size 151x19; Text 'Alarm Off Hysteresis'
   IOField "delay_startsrm_tm_sp_4" at 48,316 size 60x20; Authorization "User administration"; FormatPattern 999
      Unit <- ".Unit"
      ProcessValue <- ".FP_PARAM.Alarm_Hyst"
   CheckBox "Check box_33" at 4,316 size 32x20; Text0 'Text1'; Authorization "User administration"
      ProcessValue <- ".FP_EN.Hysteresis"
   TextField "output_head_24" at 9,356 size 151x19; Text 'Alarm Off Hysteresis'
   TextField "input_ack_1" at 12,384 size 180x20; Text 'LIM_H2 Limit H2'
   IOField "status_bit_1g_0g_32" at 72,384 size 20x20; FormatPattern 1; Unit  
      Appearance <- ".DQ.LIM_H2"
      ProcessValue <- ".DQ.LIM_H2"
   TextField "input_ack_2" at 12,406 size 180x20; Text 'LIM_H1 Limit H1'
   TextField "input_ack_3" at 12,432 size 180x20; Text 'LIM_L1 Limit L1'
   TextField "input_ack_4" at 12,455 size 180x20; Text 'LIM_L2 Limit L2'
   IOField "status_bit_1g_0g_33" at 72,407 size 20x20; FormatPattern 1; Unit  
      Appearance <- ".DQ.LIM_H1"
      ProcessValue <- ".DQ.LIM_H1"
   IOField "status_bit_1g_0g_34" at 72,432 size 20x20; FormatPattern 1; Unit  
      ProcessValue <- ".DQ.LIM_L1"
      Appearance <- ".DQ.LIM_L1"
   IOField "status_bit_1g_0g_1" at 72,455 size 20x20; FormatPattern 1; Unit  
      Appearance <- ".DQ.LIM_L2"
      ProcessValue <- ".DQ.LIM_L2"
   IOField "return_tm_sp_2" at 176,384 size 60x20; Authorization "User administration"; FormatPattern 9999
      Unit <- ".Unit"
      ProcessValue <- ".FP_PARAM.AuxLimit_H2_Value"
   IOField "delayed_run_tm_sp_2" at 176,408 size 60x20; Authorization "User administration"; FormatPattern 9999
      Unit <- ".Unit"
      ProcessValue <- ".FP_PARAM.AuxLimit_H1_Value"
   IOField "delay_stop_tm_sp_2" at 176,432 size 60x20; Authorization "User administration"; FormatPattern 999
      Unit <- ".Unit"
      ProcessValue <- ".FP_PARAM.AuxLimit_L1_Value"
   IOField "delay_startsrm_tm_sp_5" at 176,456 size 60x20; Authorization "User administration"; FormatPattern 999
      Unit <- ".Unit"
      ProcessValue <- ".FP_PARAM.AuxLimit_L2_Value"
   TextField "output_head_2" at 16,98 size 86x19; Text 'Input Signal'
   TextField "output_head_6" at 15,196 size 97x19; Text 'Signal Range'
   TextField "analog_text_6" at 24,221 size 100x20; Text 'Scale Min'
   IOField "ai2_min_sp_1" at 149,218 size 60x20; Authorization "User administration"; FormatPattern 9999.9; Unit  
      ProcessValue <- ".FP_PARAM.Scale_Min"
      Unit <- ".Unit"
   TextField "analog_text_10" at 24,245 size 100x20; Text 'Scale Max'
   IOField "ai2_max_sp_2" at 149,242 size 60x20; Authorization "User administration"; FormatPattern 9999.9; Unit  
      ProcessValue <- ".FP_PARAM.Scale_Max"
      Unit <- ".Unit"
   TextField "output_head_7" at 15,292 size 48x19; Text 'Result'
   TextField "input_rdy_8" at 24,124 size 36x20; Text 'IN'
   IOField "status_bit_1g_0r_16" at 152,124 size 60x20; FormatPattern 999.9; Unit  
      ProcessValue <- ".I.IN"
   TextField "input_rdy_9" at 24,148 size 80x20; Text 'SIG TYPE'
   IOField "status_bit_1g_0r_17" at 152,148 size 60x20; FormatPattern 99; Unit  
      ProcessValue <- ".I.SIG_TYPE"
   TextField "input_rdy_10" at 228,148 size 176x20; Text '0 - 0-100%; 1 - Scaled Val'
   IOField "status_bit_1g_0r_22" at 149,341 size 60x20; FormatPattern s999999999.9; Unit  
      FormatPattern <- ".Decimals"
      ProcessValue <- ".Q.PV_SCAL"
      Unit <- ".Unit"
   TextField "input_rdy_11" at 24,317 size 120x20; Text 'PV_NORM'
   IOField "status_bit_1g_0r_18" at 149,317 size 60x20; FormatPattern s999.9; Unit  %
      ProcessValue <- ".Q.PV_NORM"
   TextField "input_rdy_12" at 24,341 size 120x20; Text 'PV_SCAL'
   TextField "output_head_5" at 16,388 size 48x19; Text 'Force'
   IOField "ai2_max_sp_1" at 145,416 size 60x20; Authorization "User administration"; FormatPattern 9999.9; Unit  
      ProcessValue <- ".FP_PARAM.Force_Value"
   CheckBox "Check box_34" at 8,416 size 124x20; Text0 'Value'; Authorization "User administration"
      ProcessValue <- ".FP_EN.Force"
   TextField "output_head_8" at 16,100 size 101x19; Text 'Suppression'
   CheckBox "Check box_1" at 28,126 size 180x20; Text0 'Alarm Supression'; Authorization "User administration"
   TextField "head_9" at 20,103 size 99x19; Text 'Alarm Config'
   CheckBox "cb_En H3 Fatal Alarm" at 12,177 size 180x20; Text0 'En H3 Fatal Alarm'; Authorization "User administration"
      ProcessValue <- ".FP_EN.Alarm_H3"
   TextField "output_head_10" at 188,103 size 114x19; Text 'Alarm Config'
   CheckBox "cb_En L1 Warning" at 200,129 size 180x20; Text0 'En L1 Warning'; Authorization "User administration"
      ProcessValue <- ".FP_EN.Alarm_L1"
   CheckBox "cb_En L2 Warning" at 200,153 size 180x20; Text0 'En L2 Alarm'; Authorization "User administration"
      ProcessValue <- ".FP_EN.Alarm_L2"
   CheckBox "cb_En L3 Fatal Alarm" at 200,177 size 188x20; Text0 'En L3 Fatal Alarm'; Authorization "User administration"
      ProcessValue <- ".FP_EN.Alarm_L3"
   TextField "head_11" at 20,231 size 112x19; Text 'Alarm Handing'
   TextField "head_12" at 188,231 size 126x19; Text 'Enable Features'
   CheckBox "Check box_9" at 12,256 size 180x20; Text0 'Sup by Parent Grp'; Authorization "User administration"
      ProcessValue <- ".FP_EN.ParentSupress"
   CheckBox "Check box_10" at 12,280 size 188x20; Text0 'Sup to Par Grp'; Authorization "User administration"
      ProcessValue <- ".FP_EN.ParentSupressUnit"
   CheckBox "Check box_11" at 200,257 size 180x20; Text0 'Square Root'; Authorization "User administration"
      ProcessValue <- ".FP_EN.SquareRoot"
   CheckBox "Check box_12" at 200,281 size 180x20; Text0 'Squaring'; Authorization "User administration"
      ProcessValue <- ".FP_EN.Square"
   CheckBox "Check box_13" at 200,305 size 188x20; Text0 'Dumping'; Authorization "User administration"
      ProcessValue <- ".FP_EN.Damping"
   CheckBox "Check box_14" at 200,329 size 188x20; Text0 'Warning Open Loop'; Authorization "User administration"
      ProcessValue <- ".FP_EN.U_Range_Warn"
   CheckBox "Check box_15" at 200,353 size 188x20; Text0 'Warning Short Circiut'; Authorization "User administration"
      ProcessValue <- ".FP_EN.O_Range_Warn"
   TextField "output_head_13" at 20,304 size 152x19; Text 'Gradient Supervision'
   CheckBox "Check box_17" at 12,328 size 180x20; Text0 'En Pos Supervis'; Authorization "User administration"
      ProcessValue <- ".FP_EN.Gradient_Pos"
   CheckBox "Check box_18" at 12,352 size 180x20; Text0 'En Neg Supervis'; Authorization "User administration"
      ProcessValue <- ".FP_EN.Gradient_Neg"
   CheckBox "cb_En H1 Warning" at 12,128 size 180x20; Text0 'En H1 Warning'; Authorization "User administration"
      ProcessValue <- ".FP_EN.Alarm_H1"
   CheckBox "cb_En H2 Alarm" at 12,152 size 180x20; Text0 'En H2 Alarm'; Authorization "User administration"
      ProcessValue <- ".FP_EN.Alarm_H2"
   CheckBox "Check box_8" at 12,375 size 180x20; Text0 'En RateOfChng Warn'; Authorization "User administration"
      ProcessValue <- ".FP_EN.ROC_Warn"
   TextField "output_head_14" at 20,102 size 192x19; Text 'Under Range (Open Loop)'
   TextField "output_head_9" at 20,188 size 193x19; Text 'Over Range (Short Circuit)'
   TextField "output_head_11" at 20,276 size 74x19; Text 'Damping'
   TextField "input_ack_5" at 59,132 size 152x20; Text 'Signal Under Range'
   IOField "status_bit_1g_0g_2" at 32,132 size 20x20; FormatPattern 1; Unit  
      ProcessValue <- ".DI.U_RANGE"
      Appearance <- ".DI.U_RANGE"
   IOField "OpenLoopDelay_Pre_tm_sp_1" at 195,132 size 60x20; Authorization "User administration"; FormatPattern 9999; Unit  s
      ProcessValue <- ".FP_PARAM.OpenLoopDelay_Pre"
   TextField "input_ack_8" at 55,220 size 152x20; Text 'Signal Under Range'
   IOField "status_bit_1g_0g_4" at 28,220 size 20x20; FormatPattern 1; Unit  
      Appearance <- ".DI.O_RANGE"
      ProcessValue <- ".DI.O_RANGE"
   IOField "OverRangeDelay_Pre_tm_sp_2" at 191,220 size 60x20; Authorization "User administration"; FormatPattern 9999; Unit  s
      ProcessValue <- ".FP_PARAM.OverRangeDelay_Pre"
   TextField "input_ack_9" at 32,308 size 152x20; Text 'Ta Ts Dumping'
   IOField "DampingTime_sp_3" at 191,308 size 60x20; Authorization "User administration"; FormatPattern 9999; Unit  s
      ProcessValue <- ".FP_PARAM.DampingTime"
   TextField "output_head_15" at 15,99 size 114x19; Text 'PLC Subroutine'
   TextField "text_16" at 24,123 size 100x20; Text 'SubRoutine'
   TextField "text_1" at 24,151 size 100x20; Text 'Version'
   IOField "iof_vers" at 136,151 size 60x20; FormatPattern 9999; Unit  
      ProcessValue <- "[0]"
   TextField "text_2" at 24,179 size 100x20; Text 'Build'
   IOField "iof_build" at 136,179 size 60x20; FormatPattern 9999; Unit  
      ProcessValue <- "[1]"
   TextField "text_3" at 24,207 size 100x20; Text 'IOSys'
   TextField "output_head_19" at 16,259 size 106x19; Text 'PLC Reference'
   TextField "text_6" at 24,287 size 100x20; Text 'DB'
   IOField "iof_db" at 136,287 size 60x20; FormatPattern 9999; Unit  
      ProcessValue <- ".BlockInfo[2]"
   TextField "output_head_20" at 16,323 size 51x19; Text 'EcsRef'
   TextField "output_head_21" at 16,443 size 79x19; Text 'ParentInfo'
   TextField "text_7" at 24,351 size 100x20; Text 'FP Name'
   TextField "text_8" at 24,379 size 100x20; Text 'Blk Alg Ver'
   TextField "text_9" at 24,407 size 100x20; Text 'Status Alg Ver'
   IOField "parent_info" at 24,471 size 380x20; FormatPattern *; Unit  
      ProcessValue <- ".ParentInfo"
   TextField "interlockl_head_1" at 10,100 size 52x22; Text 'Trend'
   OnlineTrendControl "trend_01" at 12,124 size 392x364
      TrendTagName <- ".trend_tag_name"

VB script "layer_vis_change"
   'Tip:
   ' 1. Use the <CTRL+SPACE> or <CTRL+I> shortcut to open a list of all objects and functions
   ' 2. Write the code using the HMI Runtime object.
   '  Example: HmiRuntime.Screens("Screen_1").
   ' 3. Use the <CTRL+J> shortcut to create an object reference.
   'Write the code as of this position:
   'Please replace all sequences which are enclosed with '_' by your own code.
   
   If (Layers(2).Visible = vbFalse) Then
   	
   	Layers(2).Visible = vbTrue
   Else
   	Layers(2).Visible = vbFalse
   End If

VB script "VBFunction_1"
   'Tip:
   ' 1. Use the <CTRL+SPACE> or <CTRL+I> shortcut to open a list of all objects and functions
   ' 2. Write the code using the HMI Runtime object.
   '  Example: HmiRuntime.Screens("Screen_1").
   ' 3. Use the <CTRL+J> shortcut to create an object reference.
   'Write the code as of this position:
   
   
    
   'VBS142
   
   'Call getMousePos()
   
   Dim objRectangle, objScreenWindow, objText
   
   Set objRectangle = HMIRuntime.Screens("Main.screen_window1").ScreenItems("Rectangle")
   
   objRectangle.BackColor = RGB(255,0,0)
   
   Set objText = HMIRuntime.Screens("Main.screen_window1").ScreenItems("header_txt")
   objText.Text = "asdadasdasdasdasdas"
   'HMIRuntime.Screens("Main.screen_window1").Activate
    
   Set objScreenWindow = HMIRuntime.Screens("Main.screen_window1")
   MsgBox "Screen width before changing: " & objScreenWindow.Width
   
   
   
   'Dim objRectangle2
   '
   'Set objRectangle2 = HMIRuntime.Screens("screen_window1.screen_window2").ScreenItems("Rectangle1")
   '
   'objRectangle2.BackColor = RGB(255,159,0)
   
   'HMIRuntime.ActiveScreen.
   HMIRuntime.Trace "Customized error message"
   '

VB script "chk_popup_win_pos"
   ' Проверка координат для открытия попап окна
   ' Если окно выходит за пределы экрана то позиция корректируется
   
   ' Размер основного экрана 
   Dim m_scrn_width,  m_scrn_hight
   ' Размер popup окна
   Dim pop_win_width, pop_win_high :  pop_win_width = 500 : pop_win_high = 500
   
   HMIRuntime.Trace "1. x: " + CStr(x) + " y: " + CStr(y) + vbCrLf
   ' Размер основного экрана 
   m_scrn_width = HMIRuntime.ActiveScreen.Width
   m_scrn_hight = HMIRuntime.ActiveScreen.Height
   HMIRuntime.Trace "Scrn size: " + CStr(m_scrn_width) + " : " + CStr(m_scrn_hight) + vbCrLf
   
   'm_scrn_width = 1500
   'm_scrn_hight = 1000
   
   ' если popup окно выходит за рамки экрана то возвращаем 
   If x + pop_win_width > m_scrn_width  Then
   	x = x - (x + pop_win_width - m_scrn_width)
   	If x < 0 Then x = 0
   End If
   If y + pop_win_high > m_scrn_hight Then
   	y = y - (y + pop_win_high - m_scrn_hight)
   	If y < 0 Then x = 0
   End If
   HMIRuntime.Trace "2. x: " + CStr(x) + " y: " + CStr(y) + vbCrLf
   
   chk_popup_win_pos = Array(x,y)

VB script "show_popup_win"
   'Работа с popup Screen Windows ByVal scrn_win_title
   HMIRuntime.Trace "show_popup_win: " +tag_prefix + " : " + scrn_win_title + " : " + scrn_cntrl_name + vbCrLf
   
   Dim objOrdPpopupWinText 'текст на экране содержащий следующее popup окно.
   Dim item_index, i ' индекс для цикла 
   Dim item_name ' ObjectName  WindowsScreen
   Dim qty_popup_win_max ' максимально количество обрабатываемых WindowsScreen
   Dim ord_ppopup_win ' следующий  WindowScreen (popup) для загрузки экрана агрегата
   Dim qty_popup_win ' количество WindowsScreen на активном Screen
   Dim w_popup_arr(10) ' массив с объектами WindowsScreen активного Screen
   Dim pos_cursor_x, pos_cursor_y '- позиция кусора мыши
   Dim popup_win_ext : popup_win_ext = False ' окно с тегом уже открыто 
   
   ' Позиция очереди хранится на экране, в текстовом блоке "ord_ppopup_win"
   Set objOrdPpopupWinText = ScreenItems("ord_ppopup_win")
   ord_ppopup_win = -1 'следующий  WindowScreen для загрузки экрана агрегата
   qty_popup_win_max = 10
   qty_popup_win = 0
   
   ' Перебор всех WindowsScreen на активном screen с именем  "w_popup_unit" и сохранение в массив w_popup_arr
   For item_index = 1 To ScreenItems.Count
   	item_name = ScreenItems(item_index).ObjectName
   	If (InStr(1, item_name,"w_popup_unit",vbBinaryCompare) > 0) Then
   		'HMIRuntime.Trace CStr(item_index) + " : " + ScreenItems(item_index).ObjectName + " : " + ScreenItems(item_index).TagPrefix + Chr(13)+Chr(10)
   		Set w_popup_arr(qty_popup_win) = ScreenItems(item_index)
    		qty_popup_win = qty_popup_win + 1
   		If qty_popup_win > qty_popup_win_max Then Exit For
   		
   	End If	
   Next
   
   'HMIRuntime.Trace "Qty popw  " + CStr(qty_popup_win) + Chr(13)+Chr(10)
   
   ' Проверка есть ли уже открытое окно с заданным prefix (тегом) 
   ' и если да то в ord_ppopup_win помещаем его индекс
   For i=0 To qty_popup_win - 1
   	HMIRuntime.Trace "Check wins  " + CStr(i) + " " + w_popup_arr(i).TagPrefix + " | " + CStr(w_popup_arr(i).Visible) + " | " + tag_prefix + Chr(13)+Chr(10)
   	If (w_popup_arr(i).TagPrefix = tag_prefix And w_popup_arr(i).Visible = True ) Then ' 
   		ord_ppopup_win = i
   		popup_win_ext = True
   		'HMIRuntime.Trace "wins exist  " + CStr(i) + w_popup_arr(i).TagPrefix + " | " + CStr(w_popup_arr(i).Visible) +  Chr(13)+Chr(10)
   		Exit For
   	End If		
   Next
   ' Если нет открытого окна с заданным тегом (prefix)
   ' то ord_ppopup_win помещаем значение из очереди
   ' смещаем очередь на + 1
   If ord_ppopup_win < 0 Then
   	ord_ppopup_win = CInt(objOrdPpopupWinText.Text)
   	ord_ppopup_win = ord_ppopup_win + 1
   	If ord_ppopup_win > qty_popup_win - 1 Then ord_ppopup_win = 0
   	objOrdPpopupWinText.Text = 	CStr(ord_ppopup_win)
   		
   End If
   
   HMIRuntime.Trace "Screen open " + CStr(ord_ppopup_win) + Chr(13)+Chr(10)
   ' обновляем свойства выбранного WindowsScreen 
   w_popup_arr(ord_ppopup_win).TagPrefix = tag_prefix
   w_popup_arr(ord_ppopup_win).ScreenName = scrn_cntrl_name
   w_popup_arr(ord_ppopup_win).CaptionText = tag_prefix
   
   
   ' позицию курсора получает C script функция getMousePos и сохраняет в HMI  теги: cursor_pos_x & cursor_pos_y
   If pos_x =0 And pos_y = 0 Then
   	pos_cursor_x = HMIRuntime.Tags("cursor_pos_x").Read + 50
   	pos_cursor_y = HMIRuntime.Tags("cursor_pos_y").Read - 50
   Else
   	pos_cursor_x = pos_x
   	pos_cursor_y = pos_y
   End If
   
   
   w_popup_arr(ord_ppopup_win).Visible = False ' Если не скрывать-показать окно то оно не поднимется поверх остальных
   w_popup_arr(ord_ppopup_win).Visible = True
   'w_popup_arr(ord_ppopup_win).Activate
   'w_popup_arr(ord_ppopup_win).Screen.ScreenItems("header_txt").Text = scrn_win_title
   
   ' если окно с заданным тегом уже открыто то не меняем его координаты
   If popup_win_ext = False Then
   	w_popup_arr(ord_ppopup_win).Left = pos_cursor_x 'w_popup_arr(ord_ppopup_win).Left + 1
   	w_popup_arr(ord_ppopup_win).Top = pos_cursor_y' w_popup_arr(ord_ppopup_win).Top + 1
   End If

VB script "show_tab"
   'Показывает указанный слой, скрывая остальные
   'для реализации табов на попап окнах
   Dim objTabNumText 
   Dim layer_i
   Dim item_index, item_name, bt_lay_num
   
   'Set objTabNumText = ScreenItems("act_tab_txt")
   'objTabNumText.Text = CStr(layer)
   ' Скрываем слои 2-12, показываем указанный layer
   For layer_i = 2 To 12
   	Layers(layer_i).Visible = vbFalse
   Next
   Layers(layer + 1).Visible = vbTrue
   
   ' Подсветка кнопок выбора таба
   ' Перебераем все обекты на экране с именем bt_tab (кнопки переключения табов)
   ' и если номер в имени кнопки совпадает с переданным функции параметром то меняем заливку на светлую, если нет то на тёмную 
   For item_index = 1 To ScreenItems.Count
   	item_name = ScreenItems(item_index).ObjectName
   	If (InStr(1, item_name,"bt_tab",vbBinaryCompare) > 0) Then
   		bt_lay_num = CInt(Mid(item_name, 8 , 2))
   		'HMIRuntime.Trace CStr(item_index) + " : " + ScreenItems(item_index).ObjectName + " : " + Mid(item_name, 8 , 2) + Chr(13)+Chr(10)
   		If (bt_lay_num = layer) Then
   			ScreenItems(item_index).BackColor = RGB(255,255,255)
   			'MsgBox(item_name)
   		Else
   			ScreenItems(item_index).BackColor = RGB(150,150,150)	
   		End If	
   		
   	End If	
   Next		
   		
   		
*)

(* ===== HMI "HMI_RT_1" =====
system functions are stored by id; their names below are inferred from use

HMI tags "Default tag table"
   "msw_ext" : UInt, internal
   "msw_status" : UInt, internal
   "mode" : UInt, internal   // 0 -Auto, 2 - Local, 3 -Manual
   "status_lt" : UInt, internal   // 0 -Stoped; 1 - Run; 2- Starting; 3 - Stopping; 5 - Fault
   "test" : UInt, internal

text list "mode_l": 0 'A'; 2 'M'; 3 'L'

ScreenModuleEditorView "motor_ecs8" 1024x768
   Circle "motor_circ" at 40,5 size 48x48
      Appearance <- "status_lt"
   SymbolicIOField "mode" at 30,29 size 24x24; TextOn '1'; TextOff '0'; TextList "mode_l"
      Appearance <- "mode"
      ProcessValue <- "mode"
      Visibility <- "mode"
   TextField "x_sig" at 30,6 size 24x24; Text 'X'
      Visibility <- "status_lt"
   TextField "tag" at 6,55 size 115x21; Text 'TAG_NAME_XX'
      Text <- "TAG"
      Visible <- "TAG_VIS"
   TextField "M" at 56,17 size 18x27; Text 'M'
   TextField "title for pop windows" at 56,8 size 15x11; Text 'title'
      Text <- "TITLE"
   IOField "msw_event" at 44,40 size 42x10; FormatPattern FFFFFFFF
      ProcessValue <- "MSW"
      on ObjectChange: "OnObjectChange"
   TextField "parent info for pop windows" at 53,16 size 26x11; Text 'parent'
      Text <- "PARENT_INFO"
*)

(* ===== HMI "HMI_RT_1" =====
system functions are stored by id; their names below are inferred from use

HMI tags "Default tag table"
   "msw_ext" : UInt, internal
   "msw_status" : UInt, internal
   "mode" : UInt, internal   // 0 -Auto, 2 - Local, 3 -Manual
   "status_lt" : UInt, internal   // 0 -Close; 1 - Open; 2-Moving; 3 - Select; 5 - Fault
   "test" : UInt, internal

text list "mode_l": 0 'A'; 2 'M'; 3 'L'

ScreenModuleEditorView "valve_ecs8" 1024x768
   SymbolicIOField "mode" at 30,34 size 24x24; TextOn '1'; TextOff '0'; TextList "mode_l"
      Appearance <- "mode"
      ProcessValue <- "mode"
      Visibility <- "mode"
   TextField "x_sig" at 30,6 size 24x24; Text 'X'
      Visibility <- "status_lt"
   TextField "tag" at 17,55 size 115x21; Text 'TAG_NAME_XX'
      Text <- "TAG"
      Visible <- "TAG_VIS"
   Polygon "vlve" at 56,12 size 48x40
      Appearance <- "status_lt"
   TextField "title for pop windows" at 56,8 size 15x11; Text 'title'
      Text <- "TITLE"
   IOField "msw_event" at 64,40 size 42x10; FormatPattern FFFFFFFF
      ProcessValue <- "MSW"
      on ObjectChange: "OnObjectChange"
   TextField "parent info for pop windows" at 53,16 size 26x11; Text 'parent'
      Text <- "PARENT_INFO"
*)

(* ===== HMI "HMI_RT_1" =====
system functions are stored by id; their names below are inferred from use

HMI tags "Default tag table"
   "msw_ext" : UInt, internal
   "msw_status" : UInt, internal
   "mode" : UInt, internal   // 0 -Auto, 2 - Local, 3 -Manual
   "status_lt" : UInt, internal   // 0 -Stoped; 1 - Run; 2- Starting; 3 - Stopping; 5 - Fault
   "test" : UInt, internal

text list "mode_l": 0 'A'; 2 'M'; 3 'L'

ScreenModuleEditorView "motor_ecs8" 1024x768
   Circle "motor_circ" at 40,5 size 48x48
      Appearance <- "status_lt"
   SymbolicIOField "mode" at 30,29 size 24x24; TextOn '1'; TextOff '0'; TextList "mode_l"
      Appearance <- "mode"
      ProcessValue <- "mode"
      Visibility <- "mode"
   TextField "x_sig" at 30,6 size 24x24; Text 'X'
      Visibility <- "status_lt"
   TextField "tag" at 6,55 size 115x21; Text 'TAG_NAME_XX'
      Text <- "TAG"
      Visible <- "TAG_VIS"
   TextField "M" at 56,17 size 18x27; Text 'M'
   IOField "msw_event" at 44,40 size 42x10; FormatPattern FFFFFFFF
      ProcessValue <- "MSW"
      on ObjectChange: "OnObjectChange"
*)

(* ===== HMI "HMI_RT_1" =====
system functions are stored by id; their names below are inferred from use

HMI tags "Default tag table"
   "msw_ext" : UInt, internal
   "msw_status" : UInt, internal
   "mode" : UInt, internal   // 0 -Auto, 2 - Local, 3 -Manual
   "status_lt" : UInt, internal   // 0 -Close; 1 - Open; 2-Moving; 3 - Select; 5 - Fault
   "test" : UInt, internal

text list "mode_l": 0 'A'; 2 'M'; 3 'L'

